LIN {X 0,Y 121.489,Z 909.455,A -85,B 0,C 180,E1 27726.454,E2 27726.454} C_VEL
LIN {X 0,Y 85.535,Z 923.158,A -85,B 0,C 180,E1 27734,E2 27734} C_VEL
LIN {X 0,Y 52.423,Z 931.161,A -85,B 0,C 180,E1 27750.283,E2 27750.283} C_VEL
LIN {X 0,Y 33.25,Z 933.945,A -85,B 0,C 180,E1 27783.011,E2 27783.011} C_VEL
LIN {X 0,Y 33.264,Z 933.922,A -85,B 0,C 180,E1 27836.977,E2 27836.977} C_VEL
LIN {X 0,Y 58.65,Z 929.923,A -85,B 0,C 180,E1 27874.226,E2 27874.226} C_VEL
LIN {X 0,Y 92.609,Z 920.78,A -85,B 0,C 180,E1 27887.866,E2 27887.866} C_VEL
LIN {X 0,Y 124.559,Z 907.865,A -85,B 0,C 180,E1 27894.091,E2 27894.091} C_VEL
LIN {X 0,Y 86.399,Z 925.528,A -85,B 0,C 180,E1 27900.019,E2 27900.019} C_VEL
LIN {X 0,Y 54.099,Z 936.193,A -85,B 0,C 180,E1 27912.507,E2 27912.507} C_VEL
LIN {X 0,Y 28.099,Z 942.904,A -85,B 0,C 180,E1 27957.519,E2 27957.519} C_VEL
LIN {X 0,Y 26.517,Z 943.563,A -85,B 0,C 180,E1 27977.697,E2 27977.697} C_VEL
LIN {X 0,Y 24.613,Z 943.517,A -85,B 0,C 180,E1 27992.94,E2 27992.94} C_VEL
LIN {X 0,Y 21.913,Z 941.506,A -85,B 0,C 180,E1 28035.111,E2 28035.111} C_VEL
LIN {X 0,Y 52.923,Z 934.846,A -85,B 0,C 180,E1 28076.336,E2 28076.336} C_VEL
LIN {X 0,Y 91.062,Z 922.515,A -85,B 0,C 180,E1 28086.143,E2 28086.143} C_VEL
LIN {X 0,Y 91.268,Z 922.217,A -85,B 0,C 180,E1 28087.247,E2 28087.247} C_VEL
LIN {X 0,Y 55.679,Z 931.309,A -85,B 0,C 180,E1 28098.458,E2 28098.458} C_VEL
LIN {X 0,Y 26.544,Z 935.256,A -85,B 0,C 180,E1 28135.356,E2 28135.356} C_VEL
LIN {X 0,Y 26.557,Z 935.233,A -85,B 0,C 180,E1 28204.625,E2 28204.625} C_VEL
LIN {X 0,Y 55.691,Z 931.242,A -85,B 0,C 180,E1 28241.506,E2 28241.506} C_VEL
LIN {X 0,Y 91.285,Z 922.099,A -85,B 0,C 180,E1 28252.673,E2 28252.673} C_VEL
LIN {X 0,Y 91.061,Z 922.421,A -85,B 0,C 180,E1 28253.867,E2 28253.867} C_VEL
LIN {X 0,Y 52.923,Z 934.79,A -85,B 0,C 180,E1 28263.671,E2 28263.671} C_VEL
LIN {X 0,Y 21.684,Z 941.535,A -85,B 0,C 180,E1 28305.9,E2 28305.9} C_VEL
LIN {X 0,Y 19.235,Z 942.611,A -85,B 0,C 180,E1 28350,E2 28350} C_VEL
LIN {X 0,Y 21.913,Z 941.506,A -85,B 0,C 180,E1 28395.111,E2 28395.111} C_VEL
LIN {X 0,Y 28.591,Z 939.62,A -85,B 0,C 180,E1 28420.824,E2 28420.824} C_VEL
LIN {X 0,Y 43.222,Z 935.698,A -85,B 0,C 180,E1 28441.962,E2 28441.962} C_VEL
LIN {X 0,Y 45.265,Z 935.239,A -85,B 0,C 180,E1 28442.871,E2 28442.871} C_VEL
LIN {X 0,Y 60.829,Z 931.445,A -85,B 0,C 180,E1 28447.124,E2 28447.124} C_VEL
LIN {X 0,Y 60.982,Z 931.252,A -85,B 0,C 180,E1 28448.195,E2 28448.195} C_VEL
LIN {X 0,Y 32.698,Z 935.56,A -85,B 0,C 180,E1 28462.632,E2 28462.632} C_VEL
LIN {X 0,Y 14.451,Z 936.94,A -85,B 0,C 180,E1 28530,E2 28530} C_VEL
LIN {X 0,Y 32.705,Z 935.522,A -85,B 0,C 180,E1 28597.338,E2 28597.338} C_VEL
LIN {X 0,Y 60.991,Z 931.186,A -85,B 0,C 180,E1 28611.75,E2 28611.75} C_VEL
LIN {X 0,Y 60.826,Z 931.393,A -85,B 0,C 180,E1 28612.9,E2 28612.9} C_VEL
LIN {X 0,Y 23.216,Z 939.266,A -85,B 0,C 180,E1 28632.841,E2 28632.841} C_VEL
LIN {X 0,Y 11.204,Z 941.259,A -85,B 0,C 180,E1 28710,E2 28710} C_VEL
LIN {X 0,Y 30.317,Z 938.164,A -85,B 0,C 180,E1 28794.537,E2 28794.537} C_VEL
LIN {X 0,Y 45.265,Z 935.239,A -85,B 0,C 180,E1 28802.871,E2 28802.871} C_VEL
LIN {X 0,Y 39.983,Z 935.649,A -85,B 0,C 180,E1 28807.386,E2 28807.386} C_VEL
LIN {X 0,Y 12.03,Z 938,A -85,B 0,C 180,E1 28832.055,E2 28832.055} C_VEL
LIN {X 0,Y 16.337,Z 937.859,A -85,B 0,C 180,E1 28957.464,E2 28957.464} C_VEL
LIN {X 0,Y 24.424,Z 937.703,A -85,B 0,C 180,E1 28971.759,E2 28971.759} C_VEL
LIN {X 0,Y 3.181,Z 939.909,A -85,B 0,C 180,E1 29069.999,E2 29069.999} C_VEL
LIN {X 0,Y 24.458,Z 937.723,A -85,B 0,C 180,E1 29168.195,E2 29168.195} C_VEL
LIN {X 0,Y 16.333,Z 937.88,A -85,B 0,C 180,E1 29182.497,E2 29182.497} C_VEL
LIN {X 0,Y 12.03,Z 938,A -85,B 0,C 180,E1 29192.055,E2 29192.055} C_VEL
LIN {X 0,Y 10.461,Z 940,A -85,B 0,C 180,E1 29197.984,E2 29197.984} C_VEL
LIN {X 0,Y 10.461,Z 1015.5,A -85,B 0,C 180,E1 29197.984,E2 29197.984} C_VEL
LIN {X 0,Y 10.461,Z 1015.5,A -85,B 0,C 180,E1 29197.984,E2 29197.984}

QRS_NEXT_CUT()
PTP {E1 29336.846,E2 29336.846}
PTP {X 0,Y 607.911,A -85,B 0,C 180,E1 29336.846,E2 29336.846,E3 0,E4 0,E5 0,E6 0}
QRS_SPEED_INIT()
LIN {X 0,Y 607.911,Z 1015.5,A -85,B 0,C 180,E1 29336.846,E2 29336.846,E3 0,E4 0,E5 0,E6 0} C_VEL
LIN {X 0,Y 607.911,Z 365.088,A -85,B 0,C 180,E1 29336.846,E2 29336.846} C_VEL
LIN {X 0,Y 607.911,Z 357.012,A -85,B 0,C 180,E1 29336.846,E2 29336.846} C_VEL
LIN {X 0,Y 607.884,Z 355.012,A -85,B 0,C 180,E1 29336.657,E2 29336.657} C_VEL
LIN {X 0,Y 607.842,Z 355.013,A -85,B 0,C 180,E1 29333.767,E2 29333.767} C_VEL
LIN {X 0,Y 607.909,Z 355.01,A -85,B 0,C 180,E1 29330.629,E2 29330.629} C_VEL
LIN {X 0,Y 607.846,Z 355.012,A -85,B 0,C 180,E1 29327.652,E2 29327.652} C_VEL
LIN {X 0,Y 607.919,Z 355.009,A -85,B 0,C 180,E1 29324.516,E2 29324.516} C_VEL
LIN {X 0,Y 607.851,Z 355.012,A -85,B 0,C 180,E1 29321.49,E2 29321.49} C_VEL
LIN {X 0,Y 607.914,Z 355.01,A -85,B 0,C 180,E1 29318.382,E2 29318.382} C_VEL
LIN {X 0,Y 607.855,Z 355.012,A -85,B 0,C 180,E1 29315.304,E2 29315.304} C_VEL
LIN {X 0,Y 607.916,Z 355.01,A -85,B 0,C 180,E1 29312.223,E2 29312.223} C_VEL
LIN {X 0,Y 607.86,Z 355.011,A -85,B 0,C 180,E1 29309.153,E2 29309.153} C_VEL
LIN {X 0,Y 607.912,Z 355.011,A -85,B 0,C 180,E1 29306.112,E2 29306.112} C_VEL
LIN {X 0,Y 607.864,Z 355.01,A -85,B 0,C 180,E1 29303.065,E2 29303.065} C_VEL
LIN {X 0,Y 607.911,Z 355.011,A -85,B 0,C 180,E1 29299.977,E2 29299.977} C_VEL
LIN {X 0,Y 607.869,Z 355.01,A -85,B 0,C 180,E1 29296.822,E2 29296.822} C_VEL
LIN {X 0,Y 607.912,Z 355.011,A -85,B 0,C 180,E1 29293.776,E2 29293.776} C_VEL
LIN {X 0,Y 607.873,Z 355.009,A -85,B 0,C 180,E1 29290.639,E2 29290.639} C_VEL
LIN {X 0,Y 607.911,Z 355.008,A -85,B 0,C 180,E1 29287.48,E2 29287.48} C_VEL
LIN {X 0,Y 607.878,Z 355.011,A -85,B 0,C 180,E1 29284.34,E2 29284.34} C_VEL
LIN {X 0,Y 607.911,Z 355.004,A -85,B 0,C 180,E1 29281.201,E2 29281.201} C_VEL
LIN {X 0,Y 607.906,Z 355.317,A -85,B 0,C 180,E1 29279.834,E2 29279.834} C_VEL
LIN {X 0,Y 607.918,Z 382.895,A -85,B 0,C 180,E1 29277.643,E2 29277.643} C_VEL
LIN {X 0,Y 607.919,Z 590.082,A -85,B 0,C 180,E1 29274.95,E2 29274.95} C_VEL
LIN {X 0,Y 607.915,Z 644.717,A -85,B 0,C 180,E1 29274.225,E2 29274.225} C_VEL
LIN {X 0,Y 607.905,Z 665.586,A -85,B 0,C 180,E1 29273.761,E2 29273.761} C_VEL
LIN {X 0,Y 607.913,Z 684.825,A -85,B 0,C 180,E1 29273.16,E2 29273.16} C_VEL
LIN {X 0,Y 607.91,Z 704.295,A -85,B 0,C 180,E1 29272.378,E2 29272.378} C_VEL
LIN {X 0,Y 607.918,Z 722.621,A -85,B 0,C 180,E1 29271.468,E2 29271.468} C_VEL
LIN {X 0,Y 607.917,Z 740.995,A -85,B 0,C 180,E1 29270.364,E2 29270.364} C_VEL
LIN {X 0,Y 607.913,Z 759.159,A -85,B 0,C 180,E1 29269.053,E2 29269.053} C_VEL
LIN {X 0,Y 607.918,Z 775.938,A -85,B 0,C 180,E1 29267.613,E2 29267.613} C_VEL
LIN {X 0,Y 607.909,Z 791.465,A -85,B 0,C 180,E1 29266.039,E2 29266.039} C_VEL
LIN {X 0,Y 607.916,Z 805.424,A -85,B 0,C 180,E1 29264.362,E2 29264.362} C_VEL
LIN {X 0,Y 607.915,Z 817.506,A -85,B 0,C 180,E1 29262.634,E2 29262.634} C_VEL
LIN {X 0,Y 607.905,Z 827.625,A -85,B 0,C 180,E1 29260.902,E2 29260.902} C_VEL
LIN {X 0,Y 607.901,Z 836.374,A -85,B 0,C 180,E1 29259.084,E2 29259.084} C_VEL
LIN {X 0,Y 607.9,Z 843.351,A -85,B 0,C 180,E1 29257.275,E2 29257.275} C_VEL
LIN {X 0,Y 607.901,Z 848.889,A -85,B 0,C 180,E1 29255.379,E2 29255.379} C_VEL
LIN {X 0,Y 607.9,Z 852.665,A -85,B 0,C 180,E1 29253.488,E2 29253.488} C_VEL
LIN {X 0,Y 607.903,Z 854.841,A -85,B 0,C 180,E1 29251.602,E2 29251.602} C_VEL
LIN {X 0,Y 607.904,Z 855.45,A -85,B 0,C 180,E1 29249.717,E2 29249.717} C_VEL
LIN {X 0,Y 607.913,Z 854.498,A -85,B 0,C 180,E1 29247.832,E2 29247.832} C_VEL
LIN {X 0,Y 607.916,Z 851.71,A -85,B 0,C 180,E1 29245.85,E2 29245.85} C_VEL
LIN {X 0,Y 607.916,Z 847.356,A -85,B 0,C 180,E1 29243.958,E2 29243.958} C_VEL
LIN {X 0,Y 607.912,Z 841.288,A -85,B 0,C 180,E1 29242.059,E2 29242.059} C_VEL
LIN {X 0,Y 607.907,Z 833.818,A -85,B 0,C 180,E1 29240.247,E2 29240.247} C_VEL
LIN {X 0,Y 607.904,Z 824.477,A -85,B 0,C 180,E1 29238.425,E2 29238.425} C_VEL
LIN {X 0,Y 607.905,Z 813.618,A -85,B 0,C 180,E1 29236.688,E2 29236.688} C_VEL
LIN {X 0,Y 607.911,Z 801.351,A -85,B 0,C 180,E1 29235.036,E2 29235.036} C_VEL
LIN {X 0,Y 607.918,Z 787.678,A -85,B 0,C 180,E1 29233.47,E2 29233.47} C_VEL
LIN {X 0,Y 607.912,Z 772.518,A -85,B 0,C 180,E1 29231.99,E2 29231.99} C_VEL
LIN {X 0,Y 607.918,Z 755.721,A -85,B 0,C 180,E1 29230.597,E2 29230.597} C_VEL
LIN {X 0,Y 607.917,Z 738.595,A -85,B 0,C 180,E1 29229.394,E2 29229.394} C_VEL
LIN {X 0,Y 607.918,Z 720.445,A -85,B 0,C 180,E1 29228.322,E2 29228.322} C_VEL
LIN {X 0,Y 607.914,Z 701.781,A -85,B 0,C 180,E1 29227.418,E2 29227.418} C_VEL
LIN {X 0,Y 607.914,Z 682.685,A -85,B 0,C 180,E1 29226.676,E2 29226.676} C_VEL
LIN {X 0,Y 607.906,Z 661.895,A -85,B 0,C 180,E1 29226.058,E2 29226.058} C_VEL
LIN {X 0,Y 607.914,Z 642.161,A -85,B 0,C 180,E1 29225.645,E2 29225.645} C_VEL
LIN {X 0,Y 607.916,Z 383.636,A -85,B 0,C 180,E1 29222.289,E2 29222.289} C_VEL
LIN {X 0,Y 607.918,Z 379.216,A -85,B 0,C 180,E1 29221.988,E2 29221.988} C_VEL
LIN {X 0,Y 607.906,Z 355.369,A -85,B 0,C 180,E1 29220.088,E2 29220.088} C_VEL
LIN {X 0,Y 607.885,Z 355.008,A -85,B 0,C 180,E1 29219.674,E2 29219.674} C_VEL
LIN {X 0,Y 607.906,Z 355.01,A -85,B 0,C 180,E1 29216.501,E2 29216.501} C_VEL
LIN {X 0,Y 607.881,Z 355.009,A -85,B 0,C 180,E1 29213.387,E2 29213.387} C_VEL
LIN {X 0,Y 607.908,Z 355.011,A -85,B 0,C 180,E1 29210.227,E2 29210.227} C_VEL
LIN {X 0,Y 607.876,Z 355.009,A -85,B 0,C 180,E1 29207.189,E2 29207.189} C_VEL
LIN {X 0,Y 607.911,Z 355.011,A -85,B 0,C 180,E1 29204.054,E2 29204.054} C_VEL
LIN {X 0,Y 607.875,Z 355.009,A -85,B 0,C 180,E1 29200.893,E2 29200.893} C_VEL
LIN {X 0,Y 607.917,Z 355.013,A -85,B 0,C 180,E1 29197.717,E2 29197.717} C_VEL
LIN {X 0,Y 607.875,Z 355.008,A -85,B 0,C 180,E1 29194.574,E2 29194.574} C_VEL
LIN {X 0,Y 607.892,Z 355.013,A -85,B 0,C 180,E1 29191.316,E2 29191.316} C_VEL
LIN {X 0,Y 607.88,Z 355.008,A -85,B 0,C 180,E1 29188.276,E2 29188.276} C_VEL
LIN {X 0,Y 607.875,Z 355.013,A -85,B 0,C 180,E1 29185.007,E2 29185.007} C_VEL
LIN {X 0,Y 607.892,Z 355.008,A -85,B 0,C 180,E1 29181.94,E2 29181.94} C_VEL
LIN {X 0,Y 607.863,Z 355.012,A -85,B 0,C 180,E1 29178.709,E2 29178.709} C_VEL
LIN {X 0,Y 607.889,Z 355.009,A -85,B 0,C 180,E1 29175.747,E2 29175.747} C_VEL
LIN {X 0,Y 607.858,Z 355.013,A -85,B 0,C 180,E1 29172.54,E2 29172.54} C_VEL
LIN {X 0,Y 607.874,Z 355.01,A -85,B 0,C 180,E1 29169.659,E2 29169.659} C_VEL
LIN {X 0,Y 607.856,Z 355.013,A -85,B 0,C 180,E1 29166.422,E2 29166.422} C_VEL
LIN {X 0,Y 607.86,Z 355.011,A -85,B 0,C 180,E1 29163.584,E2 29163.584} C_VEL
LIN {X 0,Y 607.853,Z 355.014,A -85,B 0,C 180,E1 29160.283,E2 29160.283} C_VEL
LIN {X 0,Y 607.845,Z 355.012,A -85,B 0,C 180,E1 29157.549,E2 29157.549} C_VEL
LIN {X 0,Y 607.864,Z 355.014,A -85,B 0,C 180,E1 29154.299,E2 29154.299} C_VEL
LIN {X 0,Y 607.834,Z 355.014,A -85,B 0,C 180,E1 29151.487,E2 29151.487} C_VEL
LIN {X 0,Y 607.898,Z 355.015,A -85,B 0,C 180,E1 29148.424,E2 29148.424} C_VEL
LIN {X 0,Y 607.825,Z 355.014,A -85,B 0,C 180,E1 29145.521,E2 29145.521} C_VEL
LIN {X 0,Y 607.895,Z 355.015,A -85,B 0,C 180,E1 29142.532,E2 29142.532} C_VEL
LIN {X 0,Y 607.826,Z 355.015,A -85,B 0,C 180,E1 29139.49,E2 29139.49} C_VEL
LIN {X 0,Y 607.862,Z 355.014,A -85,B 0,C 180,E1 29136.646,E2 29136.646} C_VEL
LIN {X 0,Y 607.837,Z 355.014,A -85,B 0,C 180,E1 29133.422,E2 29133.422} C_VEL
LIN {X 0,Y 607.85,Z 355.014,A -85,B 0,C 180,E1 29130.648,E2 29130.648} C_VEL
LIN {X 0,Y 607.849,Z 355.013,A -85,B 0,C 180,E1 29127.349,E2 29127.349} C_VEL
LIN {X 0,Y 607.846,Z 355.013,A -85,B 0,C 180,E1 29124.619,E2 29124.619} C_VEL
LIN {X 0,Y 607.871,Z 355.011,A -85,B 0,C 180,E1 29121.373,E2 29121.373} C_VEL
LIN {X 0,Y 607.85,Z 355.013,A -85,B 0,C 180,E1 29118.479,E2 29118.479} C_VEL
LIN {X 0,Y 607.883,Z 355.011,A -85,B 0,C 180,E1 29115.253,E2 29115.253} C_VEL
LIN {X 0,Y 607.851,Z 355.012,A -85,B 0,C 180,E1 29112.391,E2 29112.391} C_VEL
LIN {X 0,Y 607.907,Z 355.002,A -85,B 0,C 180,E1 29109.224,E2 29109.224} C_VEL
LIN {X 0,Y 607.887,Z 355.304,A -85,B 0,C 180,E1 29107.84,E2 29107.84} C_VEL
LIN {X 0,Y 607.91,Z 357.762,A -85,B 0,C 180,E1 29107.654,E2 29107.654} C_VEL
LIN {X 0,Y 607.893,Z 409.406,A -85,B 0,C 180,E1 29104.798,E2 29104.798} C_VEL
LIN {X 0,Y 607.913,Z 454.921,A -85,B 0,C 180,E1 29102.376,E2 29102.376} C_VEL
LIN {X 0,Y 607.913,Z 679.75,A -85,B 0,C 180,E1 29099.342,E2 29099.342} C_VEL
LIN {X 0,Y 607.9,Z 760.832,A -85,B 0,C 180,E1 29098.245,E2 29098.245} C_VEL
LIN {X 0,Y 607.906,Z 781.277,A -85,B 0,C 180,E1 29097.804,E2 29097.804} C_VEL
LIN {X 0,Y 607.908,Z 801.875,A -85,B 0,C 180,E1 29097.207,E2 29097.207} C_VEL
LIN {X 0,Y 607.904,Z 822.631,A -85,B 0,C 180,E1 29096.415,E2 29096.415} C_VEL
LIN {X 0,Y 607.918,Z 843.787,A -85,B 0,C 180,E1 29095.419,E2 29095.419} C_VEL
LIN {X 0,Y 607.916,Z 863.097,A -85,B 0,C 180,E1 29094.332,E2 29094.332} C_VEL
LIN {X 0,Y 607.915,Z 881.589,A -85,B 0,C 180,E1 29093.094,E2 29093.094} C_VEL
LIN {X 0,Y 607.911,Z 899.77,A -85,B 0,C 180,E1 29091.678,E2 29091.678} C_VEL
LIN {X 0,Y 607.912,Z 916.668,A -85,B 0,C 180,E1 29090.154,E2 29090.154} C_VEL
LIN {X 0,Y 607.918,Z 932.477,A -85,B 0,C 180,E1 29088.506,E2 29088.506} C_VEL
LIN {X 0,Y 607.916,Z 946.401,A -85,B 0,C 180,E1 29086.818,E2 29086.818} C_VEL
LIN {X 0,Y 607.919,Z 958.909,A -85,B 0,C 180,E1 29085.061,E2 29085.061} C_VEL
LIN {X 0,Y 607.917,Z 970.422,A -85,B 0,C 180,E1 29083.176,E2 29083.176} C_VEL
LIN {X 0,Y 607.903,Z 980.064,A -85,B 0,C 180,E1 29081.286,E2 29081.286} C_VEL
LIN {X 0,Y 607.896,Z 988.387,A -85,B 0,C 180,E1 29079.296,E2 29079.296} C_VEL
LIN {X 0,Y 607.891,Z 994.96,A -85,B 0,C 180,E1 29077.339,E2 29077.339} C_VEL
LIN {X 0,Y 607.9,Z 999.809,A -85,B 0,C 180,E1 29075.379,E2 29075.379} C_VEL
LIN {X 0,Y 607.913,Z 1003.346,A -85,B 0,C 180,E1 29073.29,E2 29073.29} C_VEL
LIN {X 0,Y 607.911,Z 1005.21,A -85,B 0,C 180,E1 29071.225,E2 29071.225} C_VEL
LIN {X 0,Y 607.895,Z 1005.329,A -85,B 0,C 180,E1 29069.246,E2 29069.246} C_VEL
LIN {X 0,Y 607.89,Z 1003.896,A -85,B 0,C 180,E1 29067.172,E2 29067.172} C_VEL
LIN {X 0,Y 607.901,Z 1001.146,A -85,B 0,C 180,E1 29065.284,E2 29065.284} C_VEL
LIN {X 0,Y 607.916,Z 996.655,A -85,B 0,C 180,E1 29063.295,E2 29063.295} C_VEL
LIN {X 0,Y 607.908,Z 990.597,A -85,B 0,C 180,E1 29061.298,E2 29061.298} C_VEL
LIN {X 0,Y 607.908,Z 983.069,A -85,B 0,C 180,E1 29059.386,E2 29059.386} C_VEL
LIN {X 0,Y 607.909,Z 973.335,A -85,B 0,C 180,E1 29057.366,E2 29057.366} C_VEL
LIN {X 0,Y 607.916,Z 962.756,A -85,B 0,C 180,E1 29055.524,E2 29055.524} C_VEL
LIN {X 0,Y 607.913,Z 950.048,A -85,B 0,C 180,E1 29053.667,E2 29053.667} C_VEL
LIN {X 0,Y 607.905,Z 935.884,A -85,B 0,C 180,E1 29051.891,E2 29051.891} C_VEL
LIN {X 0,Y 607.909,Z 920.092,A -85,B 0,C 180,E1 29050.185,E2 29050.185} C_VEL
LIN {X 0,Y 607.914,Z 903.526,A -85,B 0,C 180,E1 29048.638,E2 29048.638} C_VEL
LIN {X 0,Y 607.916,Z 885.833,A -85,B 0,C 180,E1 29047.214,E2 29047.214} C_VEL
LIN {X 0,Y 607.915,Z 867.976,A -85,B 0,C 180,E1 29045.982,E2 29045.982} C_VEL
LIN {X 0,Y 607.918,Z 848.77,A -85,B 0,C 180,E1 29044.842,E2 29044.842} C_VEL
LIN {X 0,Y 607.899,Z 829.889,A -85,B 0,C 180,E1 29043.902,E2 29043.902} C_VEL
LIN {X 0,Y 607.916,Z 809.129,A -85,B 0,C 180,E1 29043.055,E2 29043.055} C_VEL
LIN {X 0,Y 607.914,Z 789.268,A -85,B 0,C 180,E1 29042.404,E2 29042.404} C_VEL
LIN {X 0,Y 607.898,Z 769.086,A -85,B 0,C 180,E1 29041.916,E2 29041.916} C_VEL
LIN {X 0,Y 607.908,Z 747.7,A -85,B 0,C 180,E1 29041.555,E2 29041.555} C_VEL
LIN {X 0,Y 607.893,Z 527.192,A -85,B 0,C 180,E1 29038.61,E2 29038.61} C_VEL
LIN {X 0,Y 607.916,Z 454.054,A -85,B 0,C 180,E1 29037.594,E2 29037.594} C_VEL
LIN {X 0,Y 607.917,Z 396.559,A -85,B 0,C 180,E1 29034.502,E2 29034.502} C_VEL
LIN {X 0,Y 607.895,Z 355.759,A -85,B 0,C 180,E1 29032.221,E2 29032.221} C_VEL
LIN {X 0,Y 607.875,Z 355.045,A -85,B 0,C 180,E1 29032.041,E2 29032.041} C_VEL
LIN {X 0,Y 607.864,Z 355.011,A -85,B 0,C 180,E1 29029.112,E2 29029.112} C_VEL
LIN {X 0,Y 607.864,Z 355.014,A -85,B 0,C 180,E1 29025.785,E2 29025.785} C_VEL
LIN {X 0,Y 607.859,Z 355.011,A -85,B 0,C 180,E1 29022.92,E2 29022.92} C_VEL
LIN {X 0,Y 607.863,Z 355.014,A -85,B 0,C 180,E1 29019.658,E2 29019.658} C_VEL
LIN {X 0,Y 607.846,Z 355.012,A -85,B 0,C 180,E1 29016.898,E2 29016.898} C_VEL
LIN {X 0,Y 607.891,Z 355.015,A -85,B 0,C 180,E1 29013.775,E2 29013.775} C_VEL
LIN {X 0,Y 607.836,Z 355.012,A -85,B 0,C 180,E1 29010.879,E2 29010.879} C_VEL
LIN {X 0,Y 607.906,Z 355.016,A -85,B 0,C 180,E1 29007.775,E2 29007.775} C_VEL
LIN {X 0,Y 607.829,Z 355.013,A -85,B 0,C 180,E1 29004.78,E2 29004.78} C_VEL
LIN {X 0,Y 607.903,Z 355.013,A -85,B 0,C 180,E1 29001.821,E2 29001.821} C_VEL
LIN {X 0,Y 607.826,Z 355.014,A -85,B 0,C 180,E1 28998.709,E2 28998.709} C_VEL
LIN {X 0,Y 607.871,Z 355.015,A -85,B 0,C 180,E1 28995.817,E2 28995.817} C_VEL
LIN {X 0,Y 607.832,Z 355.015,A -85,B 0,C 180,E1 28992.734,E2 28992.734} C_VEL
LIN {X 0,Y 607.831,Z 355.014,A -85,B 0,C 180,E1 28990.137,E2 28990.137} C_VEL
LIN {X 0,Y 607.88,Z 355.013,A -85,B 0,C 180,E1 28986.991,E2 28986.991} C_VEL
LIN {X 0,Y 607.832,Z 355.014,A -85,B 0,C 180,E1 28984.15,E2 28984.15} C_VEL
LIN {X 0,Y 607.919,Z 355.014,A -85,B 0,C 180,E1 28981.131,E2 28981.131} C_VEL
LIN {X 0,Y 607.838,Z 355.013,A -85,B 0,C 180,E1 28978.114,E2 28978.114} C_VEL
LIN {X 0,Y 607.884,Z 355.012,A -85,B 0,C 180,E1 28976.657,E2 28976.657} C_VEL
LIN {X 0,Y 606.825,Z 355.143,A -85,B 0,C 180,E1 28975.931,E2 28975.931} C_VEL
LIN {X 0,Y 600.412,Z 355.94,A -85,B 0,C 180,E1 28973.894,E2 28973.894} C_VEL
LIN {X 0,Y 599.929,Z 356.002,A -85,B 0,C 180,E1 28973.364,E2 28973.364} C_VEL
LIN {X 0,Y 599.915,Z 356,A -85,B 0,C 180,E1 28970.115,E2 28970.115} C_VEL
LIN {X 0,Y 599.924,Z 356.003,A -85,B 0,C 180,E1 28967.291,E2 28967.291} C_VEL
LIN {X 0,Y 599.927,Z 355.999,A -85,B 0,C 180,E1 28964.038,E2 28964.038} C_VEL
LIN {X 0,Y 599.928,Z 356.002,A -85,B 0,C 180,E1 28961.136,E2 28961.136} C_VEL
LIN {X 0,Y 599.933,Z 355.998,A -85,B 0,C 180,E1 28957.873,E2 28957.873} C_VEL
LIN {X 0,Y 599.932,Z 356.002,A -85,B 0,C 180,E1 28954.955,E2 28954.955} C_VEL
LIN {X 0,Y 599.932,Z 355.998,A -85,B 0,C 180,E1 28951.628,E2 28951.628} C_VEL
LIN {X 0,Y 599.958,Z 356.002,A -85,B 0,C 180,E1 28948.558,E2 28948.558} C_VEL
LIN {X 0,Y 599.932,Z 355.998,A -85,B 0,C 180,E1 28945.367,E2 28945.367} C_VEL
LIN {X 0,Y 599.972,Z 356.003,A -85,B 0,C 180,E1 28942.294,E2 28942.294} C_VEL
LIN {X 0,Y 599.931,Z 355.998,A -85,B 0,C 180,E1 28939.081,E2 28939.081} C_VEL
LIN {X 0,Y 599.975,Z 355.999,A -85,B 0,C 180,E1 28935.905,E2 28935.905} C_VEL
LIN {X 0,Y 599.934,Z 355.999,A -85,B 0,C 180,E1 28932.835,E2 28932.835} C_VEL
LIN {X 0,Y 599.974,Z 356.002,A -85,B 0,C 180,E1 28929.782,E2 28929.782} C_VEL
LIN {X 0,Y 599.937,Z 355.997,A -85,B 0,C 180,E1 28926.625,E2 28926.625} C_VEL
LIN {X 0,Y 599.97,Z 356.001,A -85,B 0,C 180,E1 28923.474,E2 28923.474} C_VEL
LIN {X 0,Y 599.948,Z 356.054,A -85,B 0,C 180,E1 28920.312,E2 28920.312} C_VEL
LIN {X 0,Y 600.063,Z 356.688,A -85,B 0,C 180,E1 28920.141,E2 28920.141} C_VEL
LIN {X 0,Y 600.588,Z 359.133,A -85,B 0,C 180,E1 28919.904,E2 28919.904} C_VEL
LIN {X 0,Y 600.567,Z 383.206,A -85,B 0,C 180,E1 28917.998,E2 28917.998} C_VEL
LIN {X 0,Y 600.82,Z 389.233,A -85,B 0,C 180,E1 28917.897,E2 28917.897} C_VEL
LIN {X 0,Y 600.615,Z 644.031,A -85,B 0,C 180,E1 28914.551,E2 28914.551} C_VEL
LIN {X 0,Y 600.559,Z 664.328,A -85,B 0,C 180,E1 28914.102,E2 28914.102} C_VEL
LIN {X 0,Y 600.503,Z 683.819,A -85,B 0,C 180,E1 28913.499,E2 28913.499} C_VEL
LIN {X 0,Y 600.422,Z 703.775,A -85,B 0,C 180,E1 28912.697,E2 28912.697} C_VEL
LIN {X 0,Y 600.356,Z 721.813,A -85,B 0,C 180,E1 28911.799,E2 28911.799} C_VEL
LIN {X 0,Y 600.284,Z 740.392,A -85,B 0,C 180,E1 28910.675,E2 28910.675} C_VEL
LIN {X 0,Y 600.201,Z 757.787,A -85,B 0,C 180,E1 28909.414,E2 28909.414} C_VEL
LIN {X 0,Y 600.125,Z 773.738,A -85,B 0,C 180,E1 28908.05,E2 28908.05} C_VEL
LIN {X 0,Y 600.068,Z 788.696,A -85,B 0,C 180,E1 28906.552,E2 28906.552} C_VEL
LIN {X 0,Y 600.014,Z 802.199,A -85,B 0,C 180,E1 28904.967,E2 28904.967} C_VEL
LIN {X 0,Y 599.967,Z 814.393,A -85,B 0,C 180,E1 28903.282,E2 28903.282} C_VEL
LIN {X 0,Y 599.939,Z 825.039,A -85,B 0,C 180,E1 28901.535,E2 28901.535} C_VEL
LIN {X 0,Y 599.925,Z 834.312,A -85,B 0,C 180,E1 28899.689,E2 28899.689} C_VEL
LIN {X 0,Y 599.919,Z 841.666,A -85,B 0,C 180,E1 28897.854,E2 28897.854} C_VEL
LIN {X 0,Y 599.917,Z 847.625,A -85,B 0,C 180,E1 28895.93,E2 28895.93} C_VEL
LIN {X 0,Y 599.917,Z 851.877,A -85,B 0,C 180,E1 28894.013,E2 28894.013} C_VEL
LIN {X 0,Y 599.915,Z 854.503,A -85,B 0,C 180,E1 28892.101,E2 28892.101} C_VEL
LIN {X 0,Y 599.912,Z 855.474,A -85,B 0,C 180,E1 28890.095,E2 28890.095} C_VEL
LIN {X 0,Y 599.909,Z 854.771,A -85,B 0,C 180,E1 28888.185,E2 28888.185} C_VEL
LIN {X 0,Y 599.913,Z 852.341,A -85,B 0,C 180,E1 28886.177,E2 28886.177} C_VEL
LIN {X 0,Y 599.918,Z 848.115,A -85,B 0,C 180,E1 28884.165,E2 28884.165} C_VEL
LIN {X 0,Y 599.925,Z 842.347,A -85,B 0,C 180,E1 28882.242,E2 28882.242} C_VEL
LIN {X 0,Y 599.928,Z 834.718,A -85,B 0,C 180,E1 28880.31,E2 28880.31} C_VEL
LIN {X 0,Y 599.939,Z 825.513,A -85,B 0,C 180,E1 28878.464,E2 28878.464} C_VEL
LIN {X 0,Y 599.968,Z 814.895,A -85,B 0,C 180,E1 28876.705,E2 28876.705} C_VEL
LIN {X 0,Y 600.01,Z 802.899,A -85,B 0,C 180,E1 28875.032,E2 28875.032} C_VEL
LIN {X 0,Y 600.065,Z 789.526,A -85,B 0,C 180,E1 28873.447,E2 28873.447} C_VEL
LIN {X 0,Y 600.124,Z 774.721,A -85,B 0,C 180,E1 28871.949,E2 28871.949} C_VEL
LIN {X 0,Y 600.202,Z 758.36,A -85,B 0,C 180,E1 28870.54,E2 28870.54} C_VEL
LIN {X 0,Y 600.277,Z 740.968,A -85,B 0,C 180,E1 28869.273,E2 28869.273} C_VEL
LIN {X 0,Y 600.35,Z 722.477,A -85,B 0,C 180,E1 28868.149,E2 28868.149} C_VEL
LIN {X 0,Y 600.422,Z 704.009,A -85,B 0,C 180,E1 28867.223,E2 28867.223} C_VEL
LIN {X 0,Y 600.501,Z 684.14,A -85,B 0,C 180,E1 28866.422,E2 28866.422} C_VEL
LIN {X 0,Y 600.558,Z 664.231,A -85,B 0,C 180,E1 28865.805,E2 28865.805} C_VEL
LIN {X 0,Y 600.616,Z 644.079,A -85,B 0,C 180,E1 28865.359,E2 28865.359} C_VEL
LIN {X 0,Y 600.825,Z 387.532,A -85,B 0,C 180,E1 28861.991,E2 28861.991} C_VEL
LIN {X 0,Y 600.547,Z 383.03,A -85,B 0,C 180,E1 28861.905,E2 28861.905} C_VEL
LIN {X 0,Y 600.55,Z 358.194,A -85,B 0,C 180,E1 28859.928,E2 28859.928} C_VEL
LIN {X 0,Y 599.96,Z 356.103,A -85,B 0,C 180,E1 28859.674,E2 28859.674} C_VEL
LIN {X 0,Y 599.968,Z 356,A -85,B 0,C 180,E1 28856.525,E2 28856.525} C_VEL
LIN {X 0,Y 599.942,Z 355.997,A -85,B 0,C 180,E1 28853.374,E2 28853.374} C_VEL
LIN {X 0,Y 599.97,Z 356.001,A -85,B 0,C 180,E1 28850.198,E2 28850.198} C_VEL
LIN {X 0,Y 599.938,Z 355.998,A -85,B 0,C 180,E1 28847.163,E2 28847.163} C_VEL
LIN {X 0,Y 599.975,Z 356,A -85,B 0,C 180,E1 28843.957,E2 28843.957} C_VEL
LIN {X 0,Y 599.94,Z 355.997,A -85,B 0,C 180,E1 28840.792,E2 28840.792} C_VEL
LIN {X 0,Y 599.96,Z 356.003,A -85,B 0,C 180,E1 28837.515,E2 28837.515} C_VEL
LIN {X 0,Y 599.949,Z 355.996,A -85,B 0,C 180,E1 28834.4,E2 28834.4} C_VEL
LIN {X 0,Y 599.936,Z 356.001,A -85,B 0,C 180,E1 28831.108,E2 28831.108} C_VEL
LIN {X 0,Y 599.974,Z 355.996,A -85,B 0,C 180,E1 28827.974,E2 28827.974} C_VEL
LIN {X 0,Y 599.926,Z 356.001,A -85,B 0,C 180,E1 28824.834,E2 28824.834} C_VEL
LIN {X 0,Y 599.968,Z 355.996,A -85,B 0,C 180,E1 28821.817,E2 28821.817} C_VEL
LIN {X 0,Y 599.922,Z 356.001,A -85,B 0,C 180,E1 28818.663,E2 28818.663} C_VEL
LIN {X 0,Y 599.959,Z 355.998,A -85,B 0,C 180,E1 28815.663,E2 28815.663} C_VEL
LIN {X 0,Y 599.918,Z 356.002,A -85,B 0,C 180,E1 28812.513,E2 28812.513} C_VEL
LIN {X 0,Y 599.942,Z 355.998,A -85,B 0,C 180,E1 28809.594,E2 28809.594} C_VEL
LIN {X 0,Y 599.917,Z 356.001,A -85,B 0,C 180,E1 28806.412,E2 28806.412} C_VEL
LIN {X 0,Y 599.925,Z 356,A -85,B 0,C 180,E1 28803.536,E2 28803.536} C_VEL
LIN {X 0,Y 599.914,Z 356.003,A -85,B 0,C 180,E1 28800.287,E2 28800.287} C_VEL
LIN {X 0,Y 599.908,Z 356.001,A -85,B 0,C 180,E1 28797.517,E2 28797.517} C_VEL
LIN {X 0,Y 599.916,Z 356.003,A -85,B 0,C 180,E1 28794.213,E2 28794.213} C_VEL
LIN {X 0,Y 599.896,Z 356.003,A -85,B 0,C 180,E1 28791.47,E2 28791.47} C_VEL
LIN {X 0,Y 599.95,Z 356.004,A -85,B 0,C 180,E1 28788.366,E2 28788.366} C_VEL
LIN {X 0,Y 599.887,Z 356.003,A -85,B 0,C 180,E1 28785.423,E2 28785.423} C_VEL
LIN {X 0,Y 599.966,Z 356.004,A -85,B 0,C 180,E1 28782.344,E2 28782.344} C_VEL
LIN {X 0,Y 599.885,Z 356.004,A -85,B 0,C 180,E1 28779.308,E2 28779.308} C_VEL
LIN {X 0,Y 599.975,Z 356,A -85,B 0,C 180,E1 28776.216,E2 28776.216} C_VEL
LIN {X 0,Y 599.891,Z 356.003,A -85,B 0,C 180,E1 28773.148,E2 28773.148} C_VEL
LIN {X 0,Y 599.971,Z 356.001,A -85,B 0,C 180,E1 28770.114,E2 28770.114} C_VEL
LIN {X 0,Y 599.899,Z 356.003,A -85,B 0,C 180,E1 28767.088,E2 28767.088} C_VEL
LIN {X 0,Y 599.947,Z 356.002,A -85,B 0,C 180,E1 28764.2,E2 28764.2} C_VEL
LIN {X 0,Y 599.909,Z 356.001,A -85,B 0,C 180,E1 28761.073,E2 28761.073} C_VEL
LIN {X 0,Y 599.938,Z 356.003,A -85,B 0,C 180,E1 28758.151,E2 28758.151} C_VEL
LIN {X 0,Y 599.916,Z 356.001,A -85,B 0,C 180,E1 28754.901,E2 28754.901} C_VEL
LIN {X 0,Y 599.947,Z 356.001,A -85,B 0,C 180,E1 28751.931,E2 28751.931} C_VEL
LIN {X 0,Y 599.918,Z 355.984,A -85,B 0,C 180,E1 28748.678,E2 28748.678} C_VEL
LIN {X 0,Y 599.959,Z 356.307,A -85,B 0,C 180,E1 28748.369,E2 28748.369} C_VEL
LIN {X 0,Y 601.251,Z 359.782,A -85,B 0,C 180,E1 28748.03,E2 28748.03} C_VEL
LIN {X 0,Y 601.05,Z 411.517,A -85,B 0,C 180,E1 28745.136,E2 28745.136} C_VEL
LIN {X 0,Y 601.04,Z 455.306,A -85,B 0,C 180,E1 28742.785,E2 28742.785} C_VEL
LIN {X 0,Y 600.971,Z 648.635,A -85,B 0,C 180,E1 28740.135,E2 28740.135} C_VEL
LIN {X 0,Y 600.843,Z 761.046,A -85,B 0,C 180,E1 28738.604,E2 28738.604} C_VEL
LIN {X 0,Y 600.786,Z 782.005,A -85,B 0,C 180,E1 28738.144,E2 28738.144} C_VEL
LIN {X 0,Y 600.712,Z 802.614,A -85,B 0,C 180,E1 28737.533,E2 28737.533} C_VEL
LIN {X 0,Y 600.636,Z 822.634,A -85,B 0,C 180,E1 28736.76,E2 28736.76} C_VEL
LIN {X 0,Y 600.539,Z 843.935,A -85,B 0,C 180,E1 28735.746,E2 28735.746} C_VEL
LIN {X 0,Y 600.444,Z 863.142,A -85,B 0,C 180,E1 28734.651,E2 28734.651} C_VEL
LIN {X 0,Y 600.354,Z 881.419,A -85,B 0,C 180,E1 28733.414,E2 28733.414} C_VEL
LIN {X 0,Y 600.249,Z 899.294,A -85,B 0,C 180,E1 28732.009,E2 28732.009} C_VEL
LIN {X 0,Y 600.159,Z 916.161,A -85,B 0,C 180,E1 28730.477,E2 28730.477} C_VEL
LIN {X 0,Y 600.108,Z 931.646,A -85,B 0,C 180,E1 28728.852,E2 28728.852} C_VEL
LIN {X 0,Y 600.04,Z 945.57,A -85,B 0,C 180,E1 28727.152,E2 28727.152} C_VEL
LIN {X 0,Y 599.989,Z 958.91,A -85,B 0,C 180,E1 28725.265,E2 28725.265} C_VEL
LIN {X 0,Y 599.952,Z 970.216,A -85,B 0,C 180,E1 28723.393,E2 28723.393} C_VEL
LIN {X 0,Y 599.925,Z 979.847,A -85,B 0,C 180,E1 28721.484,E2 28721.484} C_VEL
LIN {X 0,Y 599.905,Z 988.111,A -85,B 0,C 180,E1 28719.497,E2 28719.497} C_VEL
LIN {X 0,Y 599.903,Z 994.585,A -85,B 0,C 180,E1 28717.566,E2 28717.566} C_VEL
LIN {X 0,Y 599.911,Z 999.604,A -85,B 0,C 180,E1 28715.547,E2 28715.547} C_VEL
LIN {X 0,Y 599.915,Z 1003.222,A -85,B 0,C 180,E1 28713.44,E2 28713.44} C_VEL
LIN {X 0,Y 599.901,Z 1005.081,A -85,B 0,C 180,E1 28711.433,E2 28711.433} C_VEL
LIN {X 0,Y 599.891,Z 1005.373,A -85,B 0,C 180,E1 28709.427,E2 28709.427} C_VEL
LIN {X 0,Y 599.896,Z 1004.233,A -85,B 0,C 180,E1 28707.421,E2 28707.421} C_VEL
LIN {X 0,Y 599.909,Z 1001.463,A -85,B 0,C 180,E1 28705.412,E2 28705.412} C_VEL
LIN {X 0,Y 599.92,Z 996.909,A -85,B 0,C 180,E1 28703.301,E2 28703.301} C_VEL
LIN {X 0,Y 599.919,Z 990.792,A -85,B 0,C 180,E1 28701.235,E2 28701.235} C_VEL
LIN {X 0,Y 599.927,Z 983.07,A -85,B 0,C 180,E1 28699.243,E2 28699.243} C_VEL
LIN {X 0,Y 599.949,Z 973.336,A -85,B 0,C 180,E1 28697.195,E2 28697.195} C_VEL
LIN {X 0,Y 599.988,Z 962.755,A -85,B 0,C 180,E1 28695.329,E2 28695.329} C_VEL
LIN {X 0,Y 600.025,Z 950.049,A -85,B 0,C 180,E1 28693.446,E2 28693.446} C_VEL
LIN {X 0,Y 600.075,Z 935.885,A -85,B 0,C 180,E1 28691.647,E2 28691.647} C_VEL
LIN {X 0,Y 600.156,Z 920.218,A -85,B 0,C 180,E1 28689.931,E2 28689.931} C_VEL
LIN {X 0,Y 600.241,Z 904.131,A -85,B 0,C 180,E1 28688.402,E2 28688.402} C_VEL
LIN {X 0,Y 600.32,Z 885.833,A -85,B 0,C 180,E1 28686.909,E2 28686.909} C_VEL
LIN {X 0,Y 600.421,Z 867.176,A -85,B 0,C 180,E1 28685.61,E2 28685.61} C_VEL
LIN {X 0,Y 600.533,Z 846.786,A -85,B 0,C 180,E1 28684.405,E2 28684.405} C_VEL
LIN {X 0,Y 600.599,Z 827.615,A -85,B 0,C 180,E1 28683.452,E2 28683.452} C_VEL
LIN {X 0,Y 600.701,Z 807.05,A -85,B 0,C 180,E1 28682.628,E2 28682.628} C_VEL
LIN {X 0,Y 600.787,Z 785.722,A -85,B 0,C 180,E1 28681.953,E2 28681.953} C_VEL
LIN {X 0,Y 600.821,Z 765.977,A -85,B 0,C 180,E1 28681.49,E2 28681.49} C_VEL
LIN {X 0,Y 600.89,Z 737.832,A -85,B 0,C 180,E1 28681.06,E2 28681.06} C_VEL
LIN {X 0,Y 601.063,Z 512.335,A -85,B 0,C 180,E1 28678.007,E2 28678.007} C_VEL
LIN {X 0,Y 600.998,Z 454.722,A -85,B 0,C 180,E1 28677.194,E2 28677.194} C_VEL
LIN {X 0,Y 601.118,Z 398.862,A -85,B 0,C 180,E1 28674.167,E2 28674.167} C_VEL
LIN {X 0,Y 601.214,Z 359.452,A -85,B 0,C 180,E1 28671.949,E2 28671.949} C_VEL
LIN {X 0,Y 599.958,Z 356.295,A -85,B 0,C 180,E1 28671.631,E2 28671.631} C_VEL
LIN {X 0,Y 599.977,Z 355.984,A -85,B 0,C 180,E1 28670.59,E2 28670.59} C_VEL
LIN {X 0,Y 599.911,Z 355.998,A -85,B 0,C 180,E1 28667.551,E2 28667.551} C_VEL
LIN {X 0,Y 599.976,Z 356,A -85,B 0,C 180,E1 28664.505,E2 28664.505} C_VEL
LIN {X 0,Y 599.909,Z 356.002,A -85,B 0,C 180,E1 28661.416,E2 28661.416} C_VEL
LIN {X 0,Y 599.955,Z 356,A -85,B 0,C 180,E1 28658.435,E2 28658.435} C_VEL
LIN {X 0,Y 599.904,Z 356.001,A -85,B 0,C 180,E1 28655.255,E2 28655.255} C_VEL
LIN {X 0,Y 599.941,Z 356.001,A -85,B 0,C 180,E1 28652.342,E2 28652.342} C_VEL
LIN {X 0,Y 599.901,Z 356.002,A -85,B 0,C 180,E1 28649.16,E2 28649.16} C_VEL
LIN {X 0,Y 599.918,Z 356.002,A -85,B 0,C 180,E1 28646.316,E2 28646.316} C_VEL
LIN {X 0,Y 599.901,Z 356.002,A -85,B 0,C 180,E1 28643.059,E2 28643.059} C_VEL
LIN {X 0,Y 599.904,Z 356.003,A -85,B 0,C 180,E1 28640.24,E2 28640.24} C_VEL
LIN {X 0,Y 599.9,Z 356.004,A -85,B 0,C 180,E1 28636.944,E2 28636.944} C_VEL
LIN {X 0,Y 599.893,Z 356.004,A -85,B 0,C 180,E1 28634.182,E2 28634.182} C_VEL
LIN {X 0,Y 599.919,Z 356.003,A -85,B 0,C 180,E1 28630.952,E2 28630.952} C_VEL
LIN {X 0,Y 599.891,Z 356.003,A -85,B 0,C 180,E1 28628.137,E2 28628.137} C_VEL
LIN {X 0,Y 599.96,Z 356.002,A -85,B 0,C 180,E1 28625.067,E2 28625.067} C_VEL
LIN {X 0,Y 599.895,Z 356.002,A -85,B 0,C 180,E1 28622.101,E2 28622.101} C_VEL
LIN {X 0,Y 599.978,Z 356.001,A -85,B 0,C 180,E1 28619.045,E2 28619.045} C_VEL
LIN {X 0,Y 599.9,Z 356.002,A -85,B 0,C 180,E1 28615.986,E2 28615.986} C_VEL
LIN {X 0,Y 599.929,Z 356.002,A -85,B 0,C 180,E1 28613.364,E2 28613.364} C_VEL
LIN {X 0,Y 598.992,Z 356.126,A -85,B 0,C 180,E1 28612.629,E2 28612.629} C_VEL
LIN {X 0,Y 592.432,Z 356.937,A -85,B 0,C 180,E1 28610.512,E2 28610.512} C_VEL
LIN {X 0,Y 591.972,Z 356.988,A -85,B 0,C 180,E1 28610.027,E2 28610.027} C_VEL
LIN {X 0,Y 592.003,Z 356.992,A -85,B 0,C 180,E1 28607.118,E2 28607.118} C_VEL
LIN {X 0,Y 591.98,Z 356.989,A -85,B 0,C 180,E1 28603.919,E2 28603.919} C_VEL
LIN {X 0,Y 592.014,Z 356.992,A -85,B 0,C 180,E1 28600.874,E2 28600.874} C_VEL
LIN {X 0,Y 591.981,Z 356.988,A -85,B 0,C 180,E1 28597.664,E2 28597.664} C_VEL
LIN {X 0,Y 592.028,Z 356.993,A -85,B 0,C 180,E1 28594.597,E2 28594.597} C_VEL
LIN {X 0,Y 591.983,Z 356.989,A -85,B 0,C 180,E1 28591.424,E2 28591.424} C_VEL
LIN {X 0,Y 592.039,Z 356.992,A -85,B 0,C 180,E1 28588.316,E2 28588.316} C_VEL
LIN {X 0,Y 591.987,Z 356.988,A -85,B 0,C 180,E1 28585.161,E2 28585.161} C_VEL
LIN {X 0,Y 592.037,Z 356.984,A -85,B 0,C 180,E1 28582.055,E2 28582.055} C_VEL
LIN {X 0,Y 591.99,Z 356.988,A -85,B 0,C 180,E1 28578.927,E2 28578.927} C_VEL
LIN {X 0,Y 592.035,Z 356.985,A -85,B 0,C 180,E1 28575.725,E2 28575.725} C_VEL
LIN {X 0,Y 591.996,Z 356.99,A -85,B 0,C 180,E1 28572.575,E2 28572.575} C_VEL
LIN {X 0,Y 592.036,Z 356.985,A -85,B 0,C 180,E1 28569.331,E2 28569.331} C_VEL
LIN {X 0,Y 592.015,Z 356.989,A -85,B 0,C 180,E1 28566.112,E2 28566.112} C_VEL
LIN {X 0,Y 592.011,Z 356.988,A -85,B 0,C 180,E1 28562.745,E2 28562.745} C_VEL
LIN {X 0,Y 592.033,Z 357.184,A -85,B 0,C 180,E1 28560.578,E2 28560.578} C_VEL
LIN {X 0,Y 593.266,Z 361.864,A -85,B 0,C 180,E1 28560.088,E2 28560.088} C_VEL
LIN {X 0,Y 593.217,Z 383.41,A -85,B 0,C 180,E1 28558.372,E2 28558.372} C_VEL
LIN {X 0,Y 593.754,Z 387.573,A -85,B 0,C 180,E1 28558.281,E2 28558.281} C_VEL
LIN {X 0,Y 593.334,Z 643.972,A -85,B 0,C 180,E1 28554.875,E2 28554.875} C_VEL
LIN {X 0,Y 593.229,Z 664.355,A -85,B 0,C 180,E1 28554.419,E2 28554.419} C_VEL
LIN {X 0,Y 593.109,Z 683.84,A -85,B 0,C 180,E1 28553.81,E2 28553.81} C_VEL
LIN {X 0,Y 592.953,Z 703.211,A -85,B 0,C 180,E1 28553.027,E2 28553.027} C_VEL
LIN {X 0,Y 592.819,Z 721.822,A -85,B 0,C 180,E1 28552.091,E2 28552.091} C_VEL
LIN {X 0,Y 592.663,Z 740.404,A -85,B 0,C 180,E1 28550.954,E2 28550.954} C_VEL
LIN {X 0,Y 592.498,Z 757.875,A -85,B 0,C 180,E1 28549.67,E2 28549.67} C_VEL
LIN {X 0,Y 592.349,Z 773.745,A -85,B 0,C 180,E1 28548.296,E2 28548.296} C_VEL
LIN {X 0,Y 592.228,Z 788.703,A -85,B 0,C 180,E1 28546.778,E2 28546.778} C_VEL
LIN {X 0,Y 592.124,Z 802.206,A -85,B 0,C 180,E1 28545.171,E2 28545.171} C_VEL
LIN {X 0,Y 592.032,Z 814.959,A -85,B 0,C 180,E1 28543.376,E2 28543.376} C_VEL
LIN {X 0,Y 591.974,Z 825.62,A -85,B 0,C 180,E1 28541.582,E2 28541.582} C_VEL
LIN {X 0,Y 591.943,Z 834.754,A -85,B 0,C 180,E1 28539.723,E2 28539.723} C_VEL
LIN {X 0,Y 591.929,Z 842.376,A -85,B 0,C 180,E1 28537.765,E2 28537.765} C_VEL
LIN {X 0,Y 591.919,Z 847.88,A -85,B 0,C 180,E1 28535.913,E2 28535.913} C_VEL
LIN {X 0,Y 591.918,Z 852.195,A -85,B 0,C 180,E1 28533.874,E2 28533.874} C_VEL
LIN {X 0,Y 591.916,Z 854.643,A -85,B 0,C 180,E1 28531.936,E2 28531.936} C_VEL
LIN {X 0,Y 591.915,Z 855.494,A -85,B 0,C 180,E1 28529.903,E2 28529.903} C_VEL
LIN {X 0,Y 591.914,Z 854.57,A -85,B 0,C 180,E1 28527.87,E2 28527.87} C_VEL
LIN {X 0,Y 591.917,Z 852.025,A -85,B 0,C 180,E1 28525.932,E2 28525.932} C_VEL
LIN {X 0,Y 591.921,Z 847.86,A -85,B 0,C 180,E1 28523.989,E2 28523.989} C_VEL
LIN {X 0,Y 591.931,Z 842.345,A -85,B 0,C 180,E1 28522.137,E2 28522.137} C_VEL
LIN {X 0,Y 591.945,Z 834.716,A -85,B 0,C 180,E1 28520.178,E2 28520.178} C_VEL
LIN {X 0,Y 591.974,Z 825.511,A -85,B 0,C 180,E1 28518.307,E2 28518.307} C_VEL
LIN {X 0,Y 592.031,Z 814.891,A -85,B 0,C 180,E1 28516.524,E2 28516.524} C_VEL
LIN {X 0,Y 592.117,Z 802.895,A -85,B 0,C 180,E1 28514.828,E2 28514.828} C_VEL
LIN {X 0,Y 592.223,Z 789.248,A -85,B 0,C 180,E1 28513.192,E2 28513.192} C_VEL
LIN {X 0,Y 592.344,Z 774.716,A -85,B 0,C 180,E1 28511.703,E2 28511.703} C_VEL
LIN {X 0,Y 592.498,Z 758.354,A -85,B 0,C 180,E1 28510.277,E2 28510.277} C_VEL
LIN {X 0,Y 592.655,Z 740.955,A -85,B 0,C 180,E1 28508.993,E2 28508.993} C_VEL
LIN {X 0,Y 592.806,Z 722.461,A -85,B 0,C 180,E1 28507.856,E2 28507.856} C_VEL
LIN {X 0,Y 592.952,Z 703.999,A -85,B 0,C 180,E1 28506.92,E2 28506.92} C_VEL
LIN {X 0,Y 593.106,Z 684.125,A -85,B 0,C 180,E1 28506.11,E2 28506.11} C_VEL
LIN {X 0,Y 593.229,Z 664.206,A -85,B 0,C 180,E1 28505.487,E2 28505.487} C_VEL
LIN {X 0,Y 593.335,Z 644.039,A -85,B 0,C 180,E1 28505.037,E2 28505.037} C_VEL
LIN {X 0,Y 593.752,Z 389.39,A -85,B 0,C 180,E1 28501.653,E2 28501.653} C_VEL
LIN {X 0,Y 593.447,Z 384.6,A -85,B 0,C 180,E1 28501.573,E2 28501.573} C_VEL
LIN {X 0,Y 593.151,Z 382.815,A -85,B 0,C 180,E1 28501.51,E2 28501.51} C_VEL
LIN {X 0,Y 593.165,Z 360.909,A -85,B 0,C 180,E1 28499.738,E2 28499.738} C_VEL
LIN {X 0,Y 592.043,Z 357.203,A -85,B 0,C 180,E1 28499.338,E2 28499.338} C_VEL
LIN {X 0,Y 592.037,Z 356.987,A -85,B 0,C 180,E1 28496.133,E2 28496.133} C_VEL
LIN {X 0,Y 592.031,Z 356.981,A -85,B 0,C 180,E1 28492.803,E2 28492.803} C_VEL
LIN {X 0,Y 592.007,Z 356.986,A -85,B 0,C 180,E1 28489.572,E2 28489.572} C_VEL
LIN {X 0,Y 592.037,Z 356.985,A -85,B 0,C 180,E1 28486.429,E2 28486.429} C_VEL
LIN {X 0,Y 591.999,Z 356.988,A -85,B 0,C 180,E1 28483.292,E2 28483.292} C_VEL
LIN {X 0,Y 592.035,Z 356.987,A -85,B 0,C 180,E1 28480.095,E2 28480.095} C_VEL
LIN {X 0,Y 591.993,Z 356.988,A -85,B 0,C 180,E1 28476.961,E2 28476.961} C_VEL
LIN {X 0,Y 592.036,Z 356.989,A -85,B 0,C 180,E1 28473.815,E2 28473.815} C_VEL
LIN {X 0,Y 591.988,Z 356.987,A -85,B 0,C 180,E1 28470.669,E2 28470.669} C_VEL
LIN {X 0,Y 592.037,Z 356.991,A -85,B 0,C 180,E1 28467.455,E2 28467.455} C_VEL
LIN {X 0,Y 591.988,Z 356.988,A -85,B 0,C 180,E1 28464.338,E2 28464.338} C_VEL
LIN {X 0,Y 592.013,Z 356.992,A -85,B 0,C 180,E1 28461.084,E2 28461.084} C_VEL
LIN {X 0,Y 591.994,Z 356.987,A -85,B 0,C 180,E1 28458.004,E2 28458.004} C_VEL
LIN {X 0,Y 591.987,Z 356.99,A -85,B 0,C 180,E1 28454.676,E2 28454.676} C_VEL
LIN {X 0,Y 592.001,Z 356.988,A -85,B 0,C 180,E1 28451.694,E2 28451.694} C_VEL
LIN {X 0,Y 591.979,Z 356.991,A -85,B 0,C 180,E1 28448.45,E2 28448.45} C_VEL
LIN {X 0,Y 591.994,Z 356.987,A -85,B 0,C 180,E1 28445.525,E2 28445.525} C_VEL
LIN {X 0,Y 591.976,Z 356.99,A -85,B 0,C 180,E1 28442.323,E2 28442.323} C_VEL
LIN {X 0,Y 591.983,Z 356.99,A -85,B 0,C 180,E1 28439.42,E2 28439.42} C_VEL
LIN {X 0,Y 591.969,Z 356.992,A -85,B 0,C 180,E1 28436.126,E2 28436.126} C_VEL
LIN {X 0,Y 591.978,Z 356.99,A -85,B 0,C 180,E1 28433.238,E2 28433.238} C_VEL
LIN {X 0,Y 591.962,Z 356.992,A -85,B 0,C 180,E1 28429.941,E2 28429.941} C_VEL
LIN {X 0,Y 591.961,Z 356.992,A -85,B 0,C 180,E1 28427.217,E2 28427.217} C_VEL
LIN {X 0,Y 591.968,Z 356.993,A -85,B 0,C 180,E1 28423.919,E2 28423.919} C_VEL
LIN {X 0,Y 591.949,Z 356.992,A -85,B 0,C 180,E1 28421.179,E2 28421.179} C_VEL
LIN {X 0,Y 591.994,Z 356.991,A -85,B 0,C 180,E1 28417.979,E2 28417.979} C_VEL
LIN {X 0,Y 591.951,Z 356.989,A -85,B 0,C 180,E1 28415.088,E2 28415.088} C_VEL
LIN {X 0,Y 592.027,Z 356.99,A -85,B 0,C 180,E1 28411.998,E2 28411.998} C_VEL
LIN {X 0,Y 591.957,Z 356.988,A -85,B 0,C 180,E1 28408.992,E2 28408.992} C_VEL
LIN {X 0,Y 592.039,Z 356.988,A -85,B 0,C 180,E1 28405.896,E2 28405.896} C_VEL
LIN {X 0,Y 591.963,Z 356.991,A -85,B 0,C 180,E1 28402.794,E2 28402.794} C_VEL
LIN {X 0,Y 592.038,Z 356.988,A -85,B 0,C 180,E1 28399.698,E2 28399.698} C_VEL
LIN {X 0,Y 591.969,Z 356.99,A -85,B 0,C 180,E1 28396.57,E2 28396.57} C_VEL
LIN {X 0,Y 592.033,Z 356.984,A -85,B 0,C 180,E1 28393.417,E2 28393.417} C_VEL
LIN {X 0,Y 591.975,Z 356.993,A -85,B 0,C 180,E1 28390.382,E2 28390.382} C_VEL
LIN {X 0,Y 592.023,Z 357.165,A -85,B 0,C 180,E1 28388.949,E2 28388.949} C_VEL
LIN {X 0,Y 592.637,Z 359.298,A -85,B 0,C 180,E1 28388.712,E2 28388.712} C_VEL
LIN {X 0,Y 594.611,Z 363.476,A -85,B 0,C 180,E1 28388.317,E2 28388.317} C_VEL
LIN {X 0,Y 594.218,Z 414.579,A -85,B 0,C 180,E1 28385.43,E2 28385.43} C_VEL
LIN {X 0,Y 594.099,Z 455.361,A -85,B 0,C 180,E1 28383.216,E2 28383.216} C_VEL
LIN {X 0,Y 594.402,Z 461.097,A -85,B 0,C 180,E1 28383.116,E2 28383.116} C_VEL
LIN {X 0,Y 593.971,Z 687.339,A -85,B 0,C 180,E1 28379.997,E2 28379.997} C_VEL
LIN {X 0,Y 593.809,Z 761.902,A -85,B 0,C 180,E1 28378.961,E2 28378.961} C_VEL
LIN {X 0,Y 593.689,Z 782.798,A -85,B 0,C 180,E1 28378.49,E2 28378.49} C_VEL
LIN {X 0,Y 593.534,Z 803.499,A -85,B 0,C 180,E1 28377.862,E2 28377.862} C_VEL
LIN {X 0,Y 593.381,Z 823.91,A -85,B 0,C 180,E1 28377.059,E2 28377.059} C_VEL
LIN {X 0,Y 593.182,Z 843.793,A -85,B 0,C 180,E1 28376.097,E2 28376.097} C_VEL
LIN {X 0,Y 593.004,Z 863.138,A -85,B 0,C 180,E1 28374.982,E2 28374.982} C_VEL
LIN {X 0,Y 592.807,Z 881.666,A -85,B 0,C 180,E1 28373.712,E2 28373.712} C_VEL
LIN {X 0,Y 592.604,Z 899.296,A -85,B 0,C 180,E1 28372.309,E2 28372.309} C_VEL
LIN {X 0,Y 592.436,Z 916.161,A -85,B 0,C 180,E1 28370.756,E2 28370.756} C_VEL
LIN {X 0,Y 592.308,Z 931.601,A -85,B 0,C 180,E1 28369.115,E2 28369.115} C_VEL
LIN {X 0,Y 592.174,Z 945.571,A -85,B 0,C 180,E1 28367.387,E2 28367.387} C_VEL
LIN {X 0,Y 592.068,Z 958.911,A -85,B 0,C 180,E1 28365.474,E2 28365.474} C_VEL
LIN {X 0,Y 592.002,Z 970.217,A -85,B 0,C 180,E1 28363.577,E2 28363.577} C_VEL
LIN {X 0,Y 591.953,Z 979.603,A -85,B 0,C 180,E1 28361.693,E2 28361.693} C_VEL
LIN {X 0,Y 591.919,Z 988.112,A -85,B 0,C 180,E1 28359.626,E2 28359.626} C_VEL
LIN {X 0,Y 591.915,Z 994.585,A -85,B 0,C 180,E1 28357.668,E2 28357.668} C_VEL
LIN {X 0,Y 591.917,Z 999.604,A -85,B 0,C 180,E1 28355.622,E2 28355.622} C_VEL
LIN {X 0,Y 591.913,Z 1003.222,A -85,B 0,C 180,E1 28353.486,E2 28353.486} C_VEL
LIN {X 0,Y 591.9,Z 1005.081,A -85,B 0,C 180,E1 28351.452,E2 28351.452} C_VEL
LIN {X 0,Y 591.891,Z 1005.373,A -85,B 0,C 180,E1 28349.42,E2 28349.42} C_VEL
LIN {X 0,Y 591.894,Z 1004.233,A -85,B 0,C 180,E1 28347.386,E2 28347.386} C_VEL
LIN {X 0,Y 591.907,Z 1001.463,A -85,B 0,C 180,E1 28345.35,E2 28345.35} C_VEL
LIN {X 0,Y 591.918,Z 996.909,A -85,B 0,C 180,E1 28343.21,E2 28343.21} C_VEL
LIN {X 0,Y 591.931,Z 990.94,A -85,B 0,C 180,E1 28341.159,E2 28341.159} C_VEL
LIN {X 0,Y 591.947,Z 983.478,A -85,B 0,C 180,E1 28339.195,E2 28339.195} C_VEL
LIN {X 0,Y 591.991,Z 973.856,A -85,B 0,C 180,E1 28337.12,E2 28337.12} C_VEL
LIN {X 0,Y 592.058,Z 963.353,A -85,B 0,C 180,E1 28335.228,E2 28335.228} C_VEL
LIN {X 0,Y 592.132,Z 951.465,A -85,B 0,C 180,E1 28333.421,E2 28333.421} C_VEL
LIN {X 0,Y 592.243,Z 937.474,A -85,B 0,C 180,E1 28331.585,E2 28331.585} C_VEL
LIN {X 0,Y 592.393,Z 922.243,A -85,B 0,C 180,E1 28329.862,E2 28329.862} C_VEL
LIN {X 0,Y 592.564,Z 905.29,A -85,B 0,C 180,E1 28328.212,E2 28328.212} C_VEL
LIN {X 0,Y 592.72,Z 887.82,A -85,B 0,C 180,E1 28326.753,E2 28326.753} C_VEL
LIN {X 0,Y 592.934,Z 868.783,A -85,B 0,C 180,E1 28325.388,E2 28325.388} C_VEL
LIN {X 0,Y 593.151,Z 849.771,A -85,B 0,C 180,E1 28324.224,E2 28324.224} C_VEL
LIN {X 0,Y 593.294,Z 829.868,A -85,B 0,C 180,E1 28323.208,E2 28323.208} C_VEL
LIN {X 0,Y 593.507,Z 808.594,A -85,B 0,C 180,E1 28322.325,E2 28322.325} C_VEL
LIN {X 0,Y 593.681,Z 787.8,A -85,B 0,C 180,E1 28321.642,E2 28321.642} C_VEL
LIN {X 0,Y 593.763,Z 767.214,A -85,B 0,C 180,E1 28321.146,E2 28321.146} C_VEL
LIN {X 0,Y 593.881,Z 739.771,A -85,B 0,C 180,E1 28320.712,E2 28320.712} C_VEL
LIN {X 0,Y 594.27,Z 515.293,A -85,B 0,C 180,E1 28317.639,E2 28317.639} C_VEL
LIN {X 0,Y 594.222,Z 456.103,A -85,B 0,C 180,E1 28316.802,E2 28316.802} C_VEL
LIN {X 0,Y 593.984,Z 452.71,A -85,B 0,C 180,E1 28316.665,E2 28316.665} C_VEL
LIN {X 0,Y 594.396,Z 393.477,A -85,B 0,C 180,E1 28313.392,E2 28313.392} C_VEL
LIN {X 0,Y 594.555,Z 363.273,A -85,B 0,C 180,E1 28311.667,E2 28311.667} C_VEL
LIN {X 0,Y 592.081,Z 357.536,A -85,B 0,C 180,E1 28311.123,E2 28311.123} C_VEL
LIN {X 0,Y 592.009,Z 357.001,A -85,B 0,C 180,E1 28310.957,E2 28310.957} C_VEL
LIN {X 0,Y 591.978,Z 356.985,A -85,B 0,C 180,E1 28307.713,E2 28307.713} C_VEL
LIN {X 0,Y 592.003,Z 356.99,A -85,B 0,C 180,E1 28304.772,E2 28304.772} C_VEL
LIN {X 0,Y 591.976,Z 356.991,A -85,B 0,C 180,E1 28301.569,E2 28301.569} C_VEL
LIN {X 0,Y 591.989,Z 356.989,A -85,B 0,C 180,E1 28298.676,E2 28298.676} C_VEL
LIN {X 0,Y 591.972,Z 356.99,A -85,B 0,C 180,E1 28295.404,E2 28295.404} C_VEL
LIN {X 0,Y 591.978,Z 356.991,A -85,B 0,C 180,E1 28292.571,E2 28292.571} C_VEL
LIN {X 0,Y 591.974,Z 356.991,A -85,B 0,C 180,E1 28289.328,E2 28289.328} C_VEL
LIN {X 0,Y 591.967,Z 356.992,A -85,B 0,C 180,E1 28286.479,E2 28286.479} C_VEL
LIN {X 0,Y 591.963,Z 356.991,A -85,B 0,C 180,E1 28283.07,E2 28283.07} C_VEL
LIN {X 0,Y 591.964,Z 356.993,A -85,B 0,C 180,E1 28280.258,E2 28280.258} C_VEL
LIN {X 0,Y 591.956,Z 356.993,A -85,B 0,C 180,E1 28276.889,E2 28276.889} C_VEL
LIN {X 0,Y 591.955,Z 356.992,A -85,B 0,C 180,E1 28274.177,E2 28274.177} C_VEL
LIN {X 0,Y 591.975,Z 356.992,A -85,B 0,C 180,E1 28270.904,E2 28270.904} C_VEL
LIN {X 0,Y 591.956,Z 356.992,A -85,B 0,C 180,E1 28268.059,E2 28268.059} C_VEL
LIN {X 0,Y 591.992,Z 356.991,A -85,B 0,C 180,E1 28264.844,E2 28264.844} C_VEL
LIN {X 0,Y 591.96,Z 356.991,A -85,B 0,C 180,E1 28261.936,E2 28261.936} C_VEL
LIN {X 0,Y 592.007,Z 356.988,A -85,B 0,C 180,E1 28258.742,E2 28258.742} C_VEL
LIN {X 0,Y 591.963,Z 356.991,A -85,B 0,C 180,E1 28255.835,E2 28255.835} C_VEL
LIN {X 0,Y 592.032,Z 356.989,A -85,B 0,C 180,E1 28252.723,E2 28252.723} C_VEL
LIN {X 0,Y 591.972,Z 356.988,A -85,B 0,C 180,E1 28250.027,E2 28250.027} C_VEL
LIN {X 0,Y 590.973,Z 357.118,A -85,B 0,C 180,E1 28249.282,E2 28249.282} C_VEL
LIN {X 0,Y 584.624,Z 357.918,A -85,B 0,C 180,E1 28247.189,E2 28247.189} C_VEL
LIN {X 0,Y 584.1,Z 357.977,A -85,B 0,C 180,E1 28246.645,E2 28246.645} C_VEL
LIN {X 0,Y 584.033,Z 357.979,A -85,B 0,C 180,E1 28243.592,E2 28243.592} C_VEL
LIN {X 0,Y 584.101,Z 357.978,A -85,B 0,C 180,E1 28240.5,E2 28240.5} C_VEL
LIN {X 0,Y 584.04,Z 357.978,A -85,B 0,C 180,E1 28237.344,E2 28237.344} C_VEL
LIN {X 0,Y 584.093,Z 357.974,A -85,B 0,C 180,E1 28234.118,E2 28234.118} C_VEL
LIN {X 0,Y 584.048,Z 357.979,A -85,B 0,C 180,E1 28231.011,E2 28231.011} C_VEL
LIN {X 0,Y 584.077,Z 357.975,A -85,B 0,C 180,E1 28227.733,E2 28227.733} C_VEL
LIN {X 0,Y 584.075,Z 357.98,A -85,B 0,C 180,E1 28224.526,E2 28224.526} C_VEL
LIN {X 0,Y 584.054,Z 357.969,A -85,B 0,C 180,E1 28221.203,E2 28221.203} C_VEL
LIN {X 0,Y 584.094,Z 357.981,A -85,B 0,C 180,E1 28218.117,E2 28218.117} C_VEL
LIN {X 0,Y 584.055,Z 357.974,A -85,B 0,C 180,E1 28214.867,E2 28214.867} C_VEL
LIN {X 0,Y 584.095,Z 357.972,A -85,B 0,C 180,E1 28211.725,E2 28211.725} C_VEL
LIN {X 0,Y 584.059,Z 357.979,A -85,B 0,C 180,E1 28208.524,E2 28208.524} C_VEL
LIN {X 0,Y 584.095,Z 357.974,A -85,B 0,C 180,E1 28205.261,E2 28205.261} C_VEL
LIN {X 0,Y 584.075,Z 357.98,A -85,B 0,C 180,E1 28202.047,E2 28202.047} C_VEL
LIN {X 0,Y 584.121,Z 358.176,A -85,B 0,C 180,E1 28200.954,E2 28200.954} C_VEL
LIN {X 0,Y 585.951,Z 364.371,A -85,B 0,C 180,E1 28200.296,E2 28200.296} C_VEL
LIN {X 0,Y 585.868,Z 383.49,A -85,B 0,C 180,E1 28198.76,E2 28198.76} C_VEL
LIN {X 0,Y 586.707,Z 388.766,A -85,B 0,C 180,E1 28198.637,E2 28198.637} C_VEL
LIN {X 0,Y 586.074,Z 643.808,A -85,B 0,C 180,E1 28195.208,E2 28195.208} C_VEL
LIN {X 0,Y 585.919,Z 664.097,A -85,B 0,C 180,E1 28194.752,E2 28194.752} C_VEL
LIN {X 0,Y 585.733,Z 683.861,A -85,B 0,C 180,E1 28194.128,E2 28194.128} C_VEL
LIN {X 0,Y 585.504,Z 703.226,A -85,B 0,C 180,E1 28193.337,E2 28193.337} C_VEL
LIN {X 0,Y 585.299,Z 721.832,A -85,B 0,C 180,E1 28192.39,E2 28192.39} C_VEL
LIN {X 0,Y 585.056,Z 740.416,A -85,B 0,C 180,E1 28191.239,E2 28191.239} C_VEL
LIN {X 0,Y 584.803,Z 757.875,A -85,B 0,C 180,E1 28189.941,E2 28189.941} C_VEL
LIN {X 0,Y 584.581,Z 773.753,A -85,B 0,C 180,E1 28188.548,E2 28188.548} C_VEL
LIN {X 0,Y 584.389,Z 788.709,A -85,B 0,C 180,E1 28187.01,E2 28187.01} C_VEL
LIN {X 0,Y 584.233,Z 802.212,A -85,B 0,C 180,E1 28185.381,E2 28185.381} C_VEL
LIN {X 0,Y 584.102,Z 814.964,A -85,B 0,C 180,E1 28183.561,E2 28183.561} C_VEL
LIN {X 0,Y 584.017,Z 825.567,A -85,B 0,C 180,E1 28181.754,E2 28181.754} C_VEL
LIN {X 0,Y 583.962,Z 834.758,A -85,B 0,C 180,E1 28179.857,E2 28179.857} C_VEL
LIN {X 0,Y 583.936,Z 842.378,A -85,B 0,C 180,E1 28177.872,E2 28177.872} C_VEL
LIN {X 0,Y 583.923,Z 847.882,A -85,B 0,C 180,E1 28175.995,E2 28175.995} C_VEL
LIN {X 0,Y 583.918,Z 852.196,A -85,B 0,C 180,E1 28173.927,E2 28173.927} C_VEL
LIN {X 0,Y 583.916,Z 854.643,A -85,B 0,C 180,E1 28171.962,E2 28171.962} C_VEL
LIN {X 0,Y 583.914,Z 855.494,A -85,B 0,C 180,E1 28169.902,E2 28169.902} C_VEL
LIN {X 0,Y 583.913,Z 854.569,A -85,B 0,C 180,E1 28167.841,E2 28167.841} C_VEL
LIN {X 0,Y 583.917,Z 852.024,A -85,B 0,C 180,E1 28165.876,E2 28165.876} C_VEL
LIN {X 0,Y 583.925,Z 847.606,A -85,B 0,C 180,E1 28163.807,E2 28163.807} C_VEL
LIN {X 0,Y 583.942,Z 841.401,A -85,B 0,C 180,E1 28161.764,E2 28161.764} C_VEL
LIN {X 0,Y 583.971,Z 833.81,A -85,B 0,C 180,E1 28159.843,E2 28159.843} C_VEL
LIN {X 0,Y 584.037,Z 824.468,A -85,B 0,C 180,E1 28157.945,E2 28157.945} C_VEL
LIN {X 0,Y 584.125,Z 813.608,A -85,B 0,C 180,E1 28156.136,E2 28156.136} C_VEL
LIN {X 0,Y 584.24,Z 801.339,A -85,B 0,C 180,E1 28154.415,E2 28154.415} C_VEL
LIN {X 0,Y 584.394,Z 787.659,A -85,B 0,C 180,E1 28152.784,E2 28152.784} C_VEL
LIN {X 0,Y 584.597,Z 772.002,A -85,B 0,C 180,E1 28151.199,E2 28151.199} C_VEL
LIN {X 0,Y 584.826,Z 755.045,A -85,B 0,C 180,E1 28149.746,E2 28149.746} C_VEL
LIN {X 0,Y 585.081,Z 736.969,A -85,B 0,C 180,E1 28148.445,E2 28148.445} C_VEL
LIN {X 0,Y 585.331,Z 718.657,A -85,B 0,C 180,E1 28147.346,E2 28147.346} C_VEL
LIN {X 0,Y 585.583,Z 699.433,A -85,B 0,C 180,E1 28146.399,E2 28146.399} C_VEL
LIN {X 0,Y 585.773,Z 679.683,A -85,B 0,C 180,E1 28145.631,E2 28145.631} C_VEL
LIN {X 0,Y 585.94,Z 659.765,A -85,B 0,C 180,E1 28145.047,E2 28145.047} C_VEL
LIN {X 0,Y 586.087,Z 638.877,A -85,B 0,C 180,E1 28144.625,E2 28144.625} C_VEL
LIN {X 0,Y 586.71,Z 387.457,A -85,B 0,C 180,E1 28141.256,E2 28141.256} C_VEL
LIN {X 0,Y 585.79,Z 382.809,A -85,B 0,C 180,E1 28141.118,E2 28141.118} C_VEL
LIN {X 0,Y 585.803,Z 363.527,A -85,B 0,C 180,E1 28139.536,E2 28139.536} C_VEL
LIN {X 0,Y 584.127,Z 358.199,A -85,B 0,C 180,E1 28138.962,E2 28138.962} C_VEL
LIN {X 0,Y 584.072,Z 357.978,A -85,B 0,C 180,E1 28135.726,E2 28135.726} C_VEL
LIN {X 0,Y 584.093,Z 357.971,A -85,B 0,C 180,E1 28132.581,E2 28132.581} C_VEL
LIN {X 0,Y 584.063,Z 357.973,A -85,B 0,C 180,E1 28129.424,E2 28129.424} C_VEL
LIN {X 0,Y 584.094,Z 357.977,A -85,B 0,C 180,E1 28126.25,E2 28126.25} C_VEL
LIN {X 0,Y 584.058,Z 357.976,A -85,B 0,C 180,E1 28123.083,E2 28123.083} C_VEL
LIN {X 0,Y 584.1,Z 357.976,A -85,B 0,C 180,E1 28119.808,E2 28119.808} C_VEL
LIN {X 0,Y 584.067,Z 357.975,A -85,B 0,C 180,E1 28116.565,E2 28116.565} C_VEL
LIN {X 0,Y 584.062,Z 357.98,A -85,B 0,C 180,E1 28113.171,E2 28113.171} C_VEL
LIN {X 0,Y 584.103,Z 357.971,A -85,B 0,C 180,E1 28109.99,E2 28109.99} C_VEL
LIN {X 0,Y 584.048,Z 357.977,A -85,B 0,C 180,E1 28106.759,E2 28106.759} C_VEL
LIN {X 0,Y 584.099,Z 357.977,A -85,B 0,C 180,E1 28103.613,E2 28103.613} C_VEL
LIN {X 0,Y 584.042,Z 357.978,A -85,B 0,C 180,E1 28100.441,E2 28100.441} C_VEL
LIN {X 0,Y 584.099,Z 357.981,A -85,B 0,C 180,E1 28097.226,E2 28097.226} C_VEL
LIN {X 0,Y 584.038,Z 357.977,A -85,B 0,C 180,E1 28094.171,E2 28094.171} C_VEL
LIN {X 0,Y 584.084,Z 357.98,A -85,B 0,C 180,E1 28090.954,E2 28090.954} C_VEL
LIN {X 0,Y 584.037,Z 357.979,A -85,B 0,C 180,E1 28087.872,E2 28087.872} C_VEL
LIN {X 0,Y 584.059,Z 357.981,A -85,B 0,C 180,E1 28084.615,E2 28084.615} C_VEL
LIN {X 0,Y 584.032,Z 357.977,A -85,B 0,C 180,E1 28081.668,E2 28081.668} C_VEL
LIN {X 0,Y 584.043,Z 357.98,A -85,B 0,C 180,E1 28078.333,E2 28078.333} C_VEL
LIN {X 0,Y 584.034,Z 357.98,A -85,B 0,C 180,E1 28075.385,E2 28075.385} C_VEL
LIN {X 0,Y 584.027,Z 357.981,A -85,B 0,C 180,E1 28072.029,E2 28072.029} C_VEL
LIN {X 0,Y 584.024,Z 357.98,A -85,B 0,C 180,E1 28069.245,E2 28069.245} C_VEL
LIN {X 0,Y 584.027,Z 357.981,A -85,B 0,C 180,E1 28065.93,E2 28065.93} C_VEL
LIN {X 0,Y 584.018,Z 357.982,A -85,B 0,C 180,E1 28063.08,E2 28063.08} C_VEL
LIN {X 0,Y 584.024,Z 357.982,A -85,B 0,C 180,E1 28059.734,E2 28059.734} C_VEL
LIN {X 0,Y 584.022,Z 357.979,A -85,B 0,C 180,E1 28056.918,E2 28056.918} C_VEL
LIN {X 0,Y 584.029,Z 357.981,A -85,B 0,C 180,E1 28053.546,E2 28053.546} C_VEL
LIN {X 0,Y 584.031,Z 357.98,A -85,B 0,C 180,E1 28050.684,E2 28050.684} C_VEL
LIN {X 0,Y 584.033,Z 357.981,A -85,B 0,C 180,E1 28047.366,E2 28047.366} C_VEL
LIN {X 0,Y 584.036,Z 357.978,A -85,B 0,C 180,E1 28044.524,E2 28044.524} C_VEL
LIN {X 0,Y 584.037,Z 357.978,A -85,B 0,C 180,E1 28041.158,E2 28041.158} C_VEL
LIN {X 0,Y 584.051,Z 357.981,A -85,B 0,C 180,E1 28038.246,E2 28038.246} C_VEL
LIN {X 0,Y 584.044,Z 357.98,A -85,B 0,C 180,E1 28034.989,E2 28034.989} C_VEL
LIN {X 0,Y 584.061,Z 357.975,A -85,B 0,C 180,E1 28032.013,E2 28032.013} C_VEL
LIN {X 0,Y 584.11,Z 358.057,A -85,B 0,C 180,E1 28029.548,E2 28029.548} C_VEL
LIN {X 0,Y 584.434,Z 359.459,A -85,B 0,C 180,E1 28029.35,E2 28029.35} C_VEL
LIN {X 0,Y 587.984,Z 367.172,A -85,B 0,C 180,E1 28028.61,E2 28028.61} C_VEL
LIN {X 0,Y 587.387,Z 418.803,A -85,B 0,C 180,E1 28025.665,E2 28025.665} C_VEL
LIN {X 0,Y 587.175,Z 455.353,A -85,B 0,C 180,E1 28023.66,E2 28023.66} C_VEL
LIN {X 0,Y 587.701,Z 460.652,A -85,B 0,C 180,E1 28023.549,E2 28023.549} C_VEL
LIN {X 0,Y 587.041,Z 686.83,A -85,B 0,C 180,E1 28020.396,E2 28020.396} C_VEL
LIN {X 0,Y 586.801,Z 762.009,A -85,B 0,C 180,E1 28019.338,E2 28019.338} C_VEL
LIN {X 0,Y 586.614,Z 783.096,A -85,B 0,C 180,E1 28018.858,E2 28018.858} C_VEL
LIN {X 0,Y 586.369,Z 804.828,A -85,B 0,C 180,E1 28018.183,E2 28018.183} C_VEL
LIN {X 0,Y 586.144,Z 825.186,A -85,B 0,C 180,E1 28017.366,E2 28017.366} C_VEL
LIN {X 0,Y 585.831,Z 845.458,A -85,B 0,C 180,E1 28016.359,E2 28016.359} C_VEL
LIN {X 0,Y 585.521,Z 865.564,A -85,B 0,C 180,E1 28015.161,E2 28015.161} C_VEL
LIN {X 0,Y 585.248,Z 884.481,A -85,B 0,C 180,E1 28013.829,E2 28013.829} C_VEL
LIN {X 0,Y 584.944,Z 902.097,A -85,B 0,C 180,E1 28012.371,E2 28012.371} C_VEL
LIN {X 0,Y 584.675,Z 918.692,A -85,B 0,C 180,E1 28010.782,E2 28010.782} C_VEL
LIN {X 0,Y 584.471,Z 934.18,A -85,B 0,C 180,E1 28009.07,E2 28009.07} C_VEL
LIN {X 0,Y 584.299,Z 948.633,A -85,B 0,C 180,E1 28007.218,E2 28007.218} C_VEL
LIN {X 0,Y 584.155,Z 961.478,A -85,B 0,C 180,E1 28005.282,E2 28005.282} C_VEL
LIN {X 0,Y 584.047,Z 972.295,A -85,B 0,C 180,E1 28003.362,E2 28003.362} C_VEL
LIN {X 0,Y 583.981,Z 981.846,A -85,B 0,C 180,E1 28001.355,E2 28001.355} C_VEL
LIN {X 0,Y 583.931,Z 989.531,A -85,B 0,C 180,E1 27999.361,E2 27999.361} C_VEL
LIN {X 0,Y 583.903,Z 995.891,A -85,B 0,C 180,E1 27997.279,E2 27997.279} C_VEL
LIN {X 0,Y 583.9,Z 1000.427,A -85,B 0,C 180,E1 27995.305,E2 27995.305} C_VEL
LIN {X 0,Y 583.908,Z 1003.559,A -85,B 0,C 180,E1 27993.239,E2 27993.239} C_VEL
LIN {X 0,Y 583.913,Z 1005.262,A -85,B 0,C 180,E1 27991.08,E2 27991.08} C_VEL
LIN {X 0,Y 583.905,Z 1005.284,A -85,B 0,C 180,E1 27989.019,E2 27989.019} C_VEL
LIN {X 0,Y 583.902,Z 1003.672,A -85,B 0,C 180,E1 27986.86,E2 27986.86} C_VEL
LIN {X 0,Y 583.897,Z 1000.633,A -85,B 0,C 180,E1 27984.794,E2 27984.794} C_VEL
LIN {X 0,Y 583.904,Z 996.147,A -85,B 0,C 180,E1 27982.82,E2 27982.82} C_VEL
LIN {X 0,Y 583.934,Z 989.888,A -85,B 0,C 180,E1 27980.739,E2 27980.739} C_VEL
LIN {X 0,Y 583.98,Z 982.595,A -85,B 0,C 180,E1 27978.829,E2 27978.829} C_VEL
LIN {X 0,Y 584.044,Z 973.338,A -85,B 0,C 180,E1 27976.841,E2 27976.841} C_VEL
LIN {X 0,Y 584.152,Z 962.462,A -85,B 0,C 180,E1 27974.875,E2 27974.875} C_VEL
LIN {X 0,Y 584.276,Z 950.052,A -85,B 0,C 180,E1 27972.987,E2 27972.987} C_VEL
LIN {X 0,Y 584.444,Z 935.886,A -85,B 0,C 180,E1 27971.137,E2 27971.137} C_VEL
LIN {X 0,Y 584.662,Z 920.218,A -85,B 0,C 180,E1 27969.375,E2 27969.375} C_VEL
LIN {X 0,Y 584.927,Z 904.134,A -85,B 0,C 180,E1 27967.807,E2 27967.807} C_VEL
LIN {X 0,Y 585.202,Z 886.345,A -85,B 0,C 180,E1 27966.318,E2 27966.318} C_VEL
LIN {X 0,Y 585.472,Z 868.302,A -85,B 0,C 180,E1 27965.021,E2 27965.021} C_VEL
LIN {X 0,Y 585.806,Z 848.781,A -85,B 0,C 180,E1 27963.822,E2 27963.822} C_VEL
LIN {X 0,Y 586.039,Z 829.869,A -85,B 0,C 180,E1 27962.849,E2 27962.849} C_VEL
LIN {X 0,Y 586.338,Z 808.524,A -85,B 0,C 180,E1 27961.955,E2 27961.955} C_VEL
LIN {X 0,Y 586.6,Z 787.542,A -85,B 0,C 180,E1 27961.261,E2 27961.261} C_VEL
LIN {X 0,Y 586.735,Z 766.893,A -85,B 0,C 180,E1 27960.76,E2 27960.76} C_VEL
LIN {X 0,Y 586.905,Z 738.98,A -85,B 0,C 180,E1 27960.319,E2 27960.319} C_VEL
LIN {X 0,Y 587.513,Z 513.637,A -85,B 0,C 180,E1 27957.197,E2 27957.197} C_VEL
LIN {X 0,Y 587.512,Z 457.432,A -85,B 0,C 180,E1 27956.392,E2 27956.392} C_VEL
LIN {X 0,Y 587.058,Z 453.765,A -85,B 0,C 180,E1 27956.278,E2 27956.278} C_VEL
LIN {X 0,Y 587.679,Z 394.639,A -85,B 0,C 180,E1 27952.971,E2 27952.971} C_VEL
LIN {X 0,Y 587.898,Z 366.776,A -85,B 0,C 180,E1 27951.36,E2 27951.36} C_VEL
LIN {X 0,Y 584.181,Z 358.475,A -85,B 0,C 180,E1 27950.547,E2 27950.547} C_VEL
LIN {X 0,Y 584.089,Z 357.957,A -85,B 0,C 180,E1 27950.324,E2 27950.324} C_VEL
LIN {X 0,Y 584.033,Z 357.971,A -85,B 0,C 180,E1 27947.322,E2 27947.322} C_VEL
LIN {X 0,Y 584.093,Z 357.975,A -85,B 0,C 180,E1 27944.163,E2 27944.163} C_VEL
LIN {X 0,Y 584.03,Z 357.979,A -85,B 0,C 180,E1 27941.102,E2 27941.102} C_VEL
LIN {X 0,Y 584.077,Z 357.982,A -85,B 0,C 180,E1 27937.9,E2 27937.9} C_VEL
LIN {X 0,Y 584.026,Z 357.977,A -85,B 0,C 180,E1 27934.876,E2 27934.876} C_VEL
LIN {X 0,Y 584.07,Z 357.977,A -85,B 0,C 180,E1 27931.705,E2 27931.705} C_VEL
LIN {X 0,Y 584.02,Z 357.979,A -85,B 0,C 180,E1 27928.756,E2 27928.756} C_VEL
LIN {X 0,Y 584.068,Z 357.976,A -85,B 0,C 180,E1 27925.556,E2 27925.556} C_VEL
LIN {X 0,Y 584.013,Z 357.979,A -85,B 0,C 180,E1 27922.657,E2 27922.657} C_VEL
LIN {X 0,Y 584.081,Z 357.98,A -85,B 0,C 180,E1 27919.5,E2 27919.5} C_VEL
LIN {X 0,Y 584.007,Z 357.982,A -85,B 0,C 180,E1 27916.511,E2 27916.511} C_VEL
LIN {X 0,Y 584.086,Z 357.983,A -85,B 0,C 180,E1 27913.462,E2 27913.462} C_VEL
LIN {X 0,Y 584.01,Z 357.981,A -85,B 0,C 180,E1 27910.356,E2 27910.356} C_VEL
LIN {X 0,Y 584.098,Z 357.979,A -85,B 0,C 180,E1 27907.277,E2 27907.277} C_VEL
LIN {X 0,Y 584.017,Z 357.981,A -85,B 0,C 180,E1 27904.123,E2 27904.123} C_VEL
LIN {X 0,Y 584.09,Z 357.98,A -85,B 0,C 180,E1 27900.981,E2 27900.981} C_VEL
LIN {X 0,Y 584.022,Z 357.978,A -85,B 0,C 180,E1 27897.939,E2 27897.939} C_VEL
LIN {X 0,Y 584.092,Z 357.976,A -85,B 0,C 180,E1 27894.794,E2 27894.794} C_VEL
LIN {X 0,Y 584.027,Z 357.98,A -85,B 0,C 180,E1 27891.731,E2 27891.731} C_VEL
LIN {X 0,Y 584.09,Z 357.977,A -85,B 0,C 180,E1 27888.546,E2 27888.546} C_VEL
LIN {X 0,Y 584.1,Z 357.977,A -85,B 0,C 180,E1 27886.645,E2 27886.645} C_VEL
LIN {X 0,Y 583.096,Z 358.098,A -85,B 0,C 180,E1 27885.889,E2 27885.889} C_VEL
LIN {X 0,Y 576.616,Z 358.904,A -85,B 0,C 180,E1 27883.769,E2 27883.769} C_VEL
LIN {X 0,Y 576.108,Z 358.969,A -85,B 0,C 180,E1 27883.217,E2 27883.217} C_VEL
LIN {X 0,Y 576.11,Z 358.966,A -85,B 0,C 180,E1 27879.855,E2 27879.855} C_VEL
LIN {X 0,Y 576.134,Z 358.969,A -85,B 0,C 180,E1 27876.799,E2 27876.799} C_VEL
LIN {X 0,Y 576.106,Z 358.965,A -85,B 0,C 180,E1 27873.51,E2 27873.51} C_VEL
LIN {X 0,Y 576.162,Z 358.967,A -85,B 0,C 180,E1 27870.358,E2 27870.358} C_VEL
LIN {X 0,Y 576.107,Z 358.967,A -85,B 0,C 180,E1 27867.131,E2 27867.131} C_VEL
LIN {X 0,Y 576.16,Z 358.965,A -85,B 0,C 180,E1 27863.959,E2 27863.959} C_VEL
LIN {X 0,Y 576.112,Z 358.958,A -85,B 0,C 180,E1 27860.822,E2 27860.822} C_VEL
LIN {X 0,Y 576.156,Z 358.962,A -85,B 0,C 180,E1 27857.663,E2 27857.663} C_VEL
LIN {X 0,Y 576.122,Z 358.964,A -85,B 0,C 180,E1 27854.497,E2 27854.497} C_VEL
LIN {X 0,Y 576.136,Z 358.957,A -85,B 0,C 180,E1 27851.122,E2 27851.122} C_VEL
LIN {X 0,Y 576.157,Z 358.962,A -85,B 0,C 180,E1 27847.851,E2 27847.851} C_VEL
LIN {X 0,Y 576.123,Z 358.966,A -85,B 0,C 180,E1 27844.572,E2 27844.572} C_VEL
LIN {X 0,Y 576.18,Z 359.148,A -85,B 0,C 180,E1 27841.351,E2 27841.351} C_VEL
LIN {X 0,Y 578.636,Z 367.328,A -85,B 0,C 180,E1 27840.471,E2 27840.471} C_VEL
LIN {X 0,Y 578.527,Z 383.472,A -85,B 0,C 180,E1 27839.162,E2 27839.162} C_VEL
LIN {X 0,Y 579.681,Z 390.146,A -85,B 0,C 180,E1 27838.998,E2 27838.998} C_VEL
LIN {X 0,Y 578.833,Z 643.744,A -85,B 0,C 180,E1 27835.547,E2 27835.547} C_VEL
LIN {X 0,Y 578.628,Z 664.091,A -85,B 0,C 180,E1 27835.086,E2 27835.086} C_VEL
LIN {X 0,Y 578.374,Z 683.881,A -85,B 0,C 180,E1 27834.455,E2 27834.455} C_VEL
LIN {X 0,Y 578.085,Z 703.238,A -85,B 0,C 180,E1 27833.655,E2 27833.655} C_VEL
LIN {X 0,Y 577.794,Z 721.841,A -85,B 0,C 180,E1 27832.697,E2 27832.697} C_VEL
LIN {X 0,Y 577.462,Z 740.427,A -85,B 0,C 180,E1 27831.532,E2 27831.532} C_VEL
LIN {X 0,Y 577.123,Z 757.639,A -85,B 0,C 180,E1 27830.238,E2 27830.238} C_VEL
LIN {X 0,Y 576.824,Z 773.761,A -85,B 0,C 180,E1 27828.806,E2 27828.806} C_VEL
LIN {X 0,Y 576.564,Z 788.715,A -85,B 0,C 180,E1 27827.248,E2 27827.248} C_VEL
LIN {X 0,Y 576.353,Z 802.219,A -85,B 0,C 180,E1 27825.597,E2 27825.597} C_VEL
LIN {X 0,Y 576.183,Z 814.97,A -85,B 0,C 180,E1 27823.751,E2 27823.751} C_VEL
LIN {X 0,Y 576.065,Z 825.572,A -85,B 0,C 180,E1 27821.918,E2 27821.918} C_VEL
LIN {X 0,Y 575.984,Z 834.761,A -85,B 0,C 180,E1 27819.995,E2 27819.995} C_VEL
LIN {X 0,Y 575.945,Z 842.379,A -85,B 0,C 180,E1 27817.982,E2 27817.982} C_VEL
LIN {X 0,Y 575.926,Z 847.884,A -85,B 0,C 180,E1 27816.078,E2 27816.078} C_VEL
LIN {X 0,Y 575.918,Z 852.197,A -85,B 0,C 180,E1 27813.981,E2 27813.981} C_VEL
LIN {X 0,Y 575.916,Z 854.643,A -85,B 0,C 180,E1 27811.989,E2 27811.989} C_VEL
LIN {X 0,Y 575.914,Z 855.494,A -85,B 0,C 180,E1 27809.9,E2 27809.9} C_VEL
LIN {X 0,Y 575.911,Z 854.568,A -85,B 0,C 180,E1 27807.811,E2 27807.811} C_VEL
LIN {X 0,Y 575.918,Z 852.024,A -85,B 0,C 180,E1 27805.819,E2 27805.819} C_VEL
LIN {X 0,Y 575.927,Z 847.605,A -85,B 0,C 180,E1 27803.721,E2 27803.721} C_VEL
LIN {X 0,Y 575.952,Z 841.581,A -85,B 0,C 180,E1 27801.701,E2 27801.701} C_VEL
LIN {X 0,Y 575.993,Z 834.266,A -85,B 0,C 180,E1 27799.802,E2 27799.802} C_VEL
LIN {X 0,Y 576.078,Z 824.988,A -85,B 0,C 180,E1 27797.878,E2 27797.878} C_VEL
LIN {X 0,Y 576.196,Z 814.245,A -85,B 0,C 180,E1 27796.044,E2 27796.044} C_VEL
LIN {X 0,Y 576.354,Z 802.111,A -85,B 0,C 180,E1 27794.3,E2 27794.3} C_VEL
LIN {X 0,Y 576.564,Z 788.58,A -85,B 0,C 180,E1 27792.647,E2 27792.647} C_VEL
LIN {X 0,Y 576.826,Z 773.599,A -85,B 0,C 180,E1 27791.088,E2 27791.088} C_VEL
LIN {X 0,Y 577.125,Z 757.683,A -85,B 0,C 180,E1 27789.676,E2 27789.676} C_VEL
LIN {X 0,Y 577.465,Z 740.171,A -85,B 0,C 180,E1 27788.36,E2 27788.36} C_VEL
LIN {X 0,Y 577.797,Z 721.53,A -85,B 0,C 180,E1 27787.195,E2 27787.195} C_VEL
LIN {X 0,Y 578.094,Z 702.846,A -85,B 0,C 180,E1 27786.237,E2 27786.237} C_VEL
LIN {X 0,Y 578.371,Z 683.757,A -85,B 0,C 180,E1 27785.45,E2 27785.45} C_VEL
LIN {X 0,Y 578.634,Z 663.248,A -85,B 0,C 180,E1 27784.802,E2 27784.802} C_VEL
LIN {X 0,Y 578.837,Z 643.026,A -85,B 0,C 180,E1 27784.352,E2 27784.352} C_VEL
LIN {X 0,Y 579.688,Z 389.03,A -85,B 0,C 180,E1 27780.897,E2 27780.897} C_VEL
LIN {X 0,Y 578.455,Z 382.817,A -85,B 0,C 180,E1 27780.717,E2 27780.717} C_VEL
LIN {X 0,Y 578.467,Z 366.341,A -85,B 0,C 180,E1 27779.346,E2 27779.346} C_VEL
LIN {X 0,Y 576.189,Z 359.231,A -85,B 0,C 180,E1 27778.579,E2 27778.579} C_VEL
LIN {X 0,Y 576.155,Z 358.967,A -85,B 0,C 180,E1 27776.951,E2 27776.951} C_VEL
LIN {X 0,Y 576.129,Z 358.964,A -85,B 0,C 180,E1 27773.596,E2 27773.596} C_VEL
LIN {X 0,Y 576.154,Z 358.966,A -85,B 0,C 180,E1 27770.401,E2 27770.401} C_VEL
LIN {X 0,Y 576.122,Z 358.967,A -85,B 0,C 180,E1 27767.233,E2 27767.233} C_VEL
LIN {X 0,Y 576.157,Z 358.961,A -85,B 0,C 180,E1 27763.96,E2 27763.96} C_VEL
LIN {X 0,Y 576.132,Z 358.964,A -85,B 0,C 180,E1 27760.683,E2 27760.683} C_VEL
LIN {X 0,Y 576.125,Z 358.968,A -85,B 0,C 180,E1 27757.278,E2 27757.278} C_VEL
LIN {X 0,Y 576.16,Z 358.962,A -85,B 0,C 180,E1 27754.093,E2 27754.093} C_VEL
LIN {X 0,Y 576.112,Z 358.965,A -85,B 0,C 180,E1 27750.912,E2 27750.912} C_VEL
LIN {X 0,Y 576.162,Z 358.966,A -85,B 0,C 180,E1 27747.716,E2 27747.716} C_VEL
LIN {X 0,Y 576.106,Z 358.966,A -85,B 0,C 180,E1 27744.507,E2 27744.507} C_VEL
LIN {X 0,Y 576.154,Z 358.971,A -85,B 0,C 180,E1 27741.266,E2 27741.266} C_VEL
LIN {X 0,Y 576.111,Z 358.965,A -85,B 0,C 180,E1 27738.099,E2 27738.099} C_VEL
LIN {X 0,Y 576.11,Z 358.968,A -85,B 0,C 180,E1 27734.678,E2 27734.678} C_VEL
LIN {X 0,Y 576.131,Z 358.966,A -85,B 0,C 180,E1 27731.614,E2 27731.614} C_VEL
LIN {X 0,Y 576.099,Z 358.969,A -85,B 0,C 180,E1 27728.383,E2 27728.383} C_VEL
LIN {X 0,Y 576.144,Z 358.963,A -85,B 0,C 180,E1 27725.278,E2 27725.278} C_VEL
LIN {X 0,Y 576.088,Z 358.966,A -85,B 0,C 180,E1 27722.089,E2 27722.089} C_VEL
LIN {X 0,Y 576.153,Z 358.968,A -85,B 0,C 180,E1 27719.006,E2 27719.006} C_VEL
LIN {X 0,Y 576.081,Z 358.97,A -85,B 0,C 180,E1 27715.82,E2 27715.82} C_VEL
LIN {X 0,Y 576.159,Z 358.967,A -85,B 0,C 180,E1 27712.722,E2 27712.722} C_VEL
LIN {X 0,Y 576.074,Z 358.969,A -85,B 0,C 180,E1 27709.601,E2 27709.601} C_VEL
LIN {X 0,Y 576.149,Z 358.971,A -85,B 0,C 180,E1 27706.451,E2 27706.451} C_VEL
LIN {X 0,Y 576.069,Z 358.971,A -85,B 0,C 180,E1 27703.359,E2 27703.359} C_VEL
LIN {X 0,Y 576.137,Z 358.972,A -85,B 0,C 180,E1 27700.22,E2 27700.22} C_VEL
LIN {X 0,Y 576.074,Z 358.968,A -85,B 0,C 180,E1 27697.121,E2 27697.121} C_VEL
LIN {X 0,Y 576.132,Z 358.97,A -85,B 0,C 180,E1 27693.956,E2 27693.956} C_VEL
LIN {X 0,Y 576.08,Z 358.969,A -85,B 0,C 180,E1 27690.924,E2 27690.924} C_VEL
LIN {X 0,Y 576.142,Z 358.969,A -85,B 0,C 180,E1 27687.807,E2 27687.807} C_VEL
LIN {X 0,Y 576.085,Z 358.965,A -85,B 0,C 180,E1 27684.815,E2 27684.815} C_VEL
LIN {X 0,Y 576.142,Z 358.966,A -85,B 0,C 180,E1 27681.59,E2 27681.59} C_VEL
LIN {X 0,Y 576.093,Z 358.969,A -85,B 0,C 180,E1 27678.565,E2 27678.565} C_VEL
LIN {X 0,Y 576.138,Z 358.967,A -85,B 0,C 180,E1 27675.344,E2 27675.344} C_VEL
LIN {X 0,Y 576.099,Z 358.962,A -85,B 0,C 180,E1 27672.324,E2 27672.324} C_VEL
LIN {X 0,Y 576.124,Z 359.083,A -85,B 0,C 180,E1 27670.141,E2 27670.141} C_VEL
LIN {X 0,Y 576.446,Z 360.415,A -85,B 0,C 180,E1 27669.946,E2 27669.946} C_VEL
LIN {X 0,Y 581.361,Z 370.567,A -85,B 0,C 180,E1 27668.93,E2 27668.93} C_VEL
LIN {X 0,Y 580.596,Z 421.125,A -85,B 0,C 180,E1 27666.013,E2 27666.013} C_VEL
LIN {X 0,Y 580.28,Z 455.281,A -85,B 0,C 180,E1 27664.116,E2 27664.116} C_VEL
LIN {X 0,Y 581.026,Z 461.704,A -85,B 0,C 180,E1 27663.972,E2 27663.972} C_VEL
LIN {X 0,Y 580.135,Z 688.102,A -85,B 0,C 180,E1 27660.779,E2 27660.779} C_VEL
LIN {X 0,Y 579.819,Z 762.116,A -85,B 0,C 180,E1 27659.725,E2 27659.725} C_VEL
LIN {X 0,Y 579.565,Z 783.356,A -85,B 0,C 180,E1 27659.236,E2 27659.236} C_VEL
LIN {X 0,Y 579.252,Z 804.824,A -85,B 0,C 180,E1 27658.561,E2 27658.561} C_VEL
LIN {X 0,Y 578.937,Z 825.189,A -85,B 0,C 180,E1 27657.736,E2 27657.736} C_VEL
LIN {X 0,Y 578.525,Z 844.792,A -85,B 0,C 180,E1 27656.755,E2 27656.755} C_VEL
LIN {X 0,Y 578.136,Z 864.753,A -85,B 0,C 180,E1 27655.56,E2 27655.56} C_VEL
LIN {X 0,Y 577.736,Z 883.814,A -85,B 0,C 180,E1 27654.21,E2 27654.21} C_VEL
LIN {X 0,Y 577.325,Z 901.713,A -85,B 0,C 180,E1 27652.717,E2 27652.717} C_VEL
LIN {X 0,Y 576.966,Z 918.825,A -85,B 0,C 180,E1 27651.059,E2 27651.059} C_VEL
LIN {X 0,Y 576.682,Z 934.181,A -85,B 0,C 180,E1 27649.337,E2 27649.337} C_VEL
LIN {X 0,Y 576.437,Z 948.634,A -85,B 0,C 180,E1 27647.461,E2 27647.461} C_VEL
LIN {X 0,Y 576.237,Z 960.838,A -85,B 0,C 180,E1 27645.6,E2 27645.6} C_VEL
LIN {X 0,Y 576.093,Z 972.297,A -85,B 0,C 180,E1 27643.55,E2 27643.55} C_VEL
LIN {X 0,Y 576.005,Z 981.847,A -85,B 0,C 180,E1 27641.514,E2 27641.514} C_VEL
LIN {X 0,Y 575.943,Z 989.235,A -85,B 0,C 180,E1 27639.577,E2 27639.577} C_VEL
LIN {X 0,Y 575.908,Z 995.891,A -85,B 0,C 180,E1 27637.381,E2 27637.381} C_VEL
LIN {X 0,Y 575.905,Z 1000.427,A -85,B 0,C 180,E1 27635.379,E2 27635.379} C_VEL
LIN {X 0,Y 575.912,Z 1003.56,A -85,B 0,C 180,E1 27633.284,E2 27633.284} C_VEL
LIN {X 0,Y 575.913,Z 1005.262,A -85,B 0,C 180,E1 27631.095,E2 27631.095} C_VEL
LIN {X 0,Y 575.907,Z 1005.284,A -85,B 0,C 180,E1 27629.006,E2 27629.006} C_VEL
LIN {X 0,Y 575.904,Z 1003.672,A -85,B 0,C 180,E1 27626.816,E2 27626.816} C_VEL
LIN {X 0,Y 575.9,Z 1000.633,A -85,B 0,C 180,E1 27624.721,E2 27624.721} C_VEL
LIN {X 0,Y 575.907,Z 996.147,A -85,B 0,C 180,E1 27622.72,E2 27622.72} C_VEL
LIN {X 0,Y 575.944,Z 989.889,A -85,B 0,C 180,E1 27620.609,E2 27620.609} C_VEL
LIN {X 0,Y 576.003,Z 982.664,A -85,B 0,C 180,E1 27618.689,E2 27618.689} C_VEL
LIN {X 0,Y 576.093,Z 973.339,A -85,B 0,C 180,E1 27616.656,E2 27616.656} C_VEL
LIN {X 0,Y 576.234,Z 962.751,A -85,B 0,C 180,E1 27614.71,E2 27614.71} C_VEL
LIN {X 0,Y 576.399,Z 950.76,A -85,B 0,C 180,E1 27612.851,E2 27612.851} C_VEL
LIN {X 0,Y 576.63,Z 936.737,A -85,B 0,C 180,E1 27610.977,E2 27610.977} C_VEL
LIN {X 0,Y 576.919,Z 921.658,A -85,B 0,C 180,E1 27609.237,E2 27609.237} C_VEL
LIN {X 0,Y 577.283,Z 904.759,A -85,B 0,C 180,E1 27607.554,E2 27607.554} C_VEL
LIN {X 0,Y 577.669,Z 886.492,A -85,B 0,C 180,E1 27606.002,E2 27606.002} C_VEL
LIN {X 0,Y 578.042,Z 867.986,A -85,B 0,C 180,E1 27604.656,E2 27604.656} C_VEL
LIN {X 0,Y 578.476,Z 848.783,A -85,B 0,C 180,E1 27603.465,E2 27603.465} C_VEL
LIN {X 0,Y 578.817,Z 829.866,A -85,B 0,C 180,E1 27602.482,E2 27602.482} C_VEL
LIN {X 0,Y 579.195,Z 808.527,A -85,B 0,C 180,E1 27601.577,E2 27601.577} C_VEL
LIN {X 0,Y 579.545,Z 787.414,A -85,B 0,C 180,E1 27600.874,E2 27600.874} C_VEL
LIN {X 0,Y 579.736,Z 766.498,A -85,B 0,C 180,E1 27600.364,E2 27600.364} C_VEL
LIN {X 0,Y 579.959,Z 737.765,A -85,B 0,C 180,E1 27599.91,E2 27599.91} C_VEL
LIN {X 0,Y 580.794,Z 511.444,A -85,B 0,C 180,E1 27596.737,E2 27596.737} C_VEL
LIN {X 0,Y 580.835,Z 458.757,A -85,B 0,C 180,E1 27595.973,E2 27595.973} C_VEL
LIN {X 0,Y 580.178,Z 453.598,A -85,B 0,C 180,E1 27595.813,E2 27595.813} C_VEL
LIN {X 0,Y 581.013,Z 394.639,A -85,B 0,C 180,E1 27592.474,E2 27592.474} C_VEL
LIN {X 0,Y 581.195,Z 370.294,A -85,B 0,C 180,E1 27591.041,E2 27591.041} C_VEL
LIN {X 0,Y 577.396,Z 362.346,A -85,B 0,C 180,E1 27590.251,E2 27590.251} C_VEL
LIN {X 0,Y 576.173,Z 359.352,A -85,B 0,C 180,E1 27589.929,E2 27589.929} C_VEL
LIN {X 0,Y 576.096,Z 358.962,A -85,B 0,C 180,E1 27589.48,E2 27589.48} C_VEL
LIN {X 0,Y 576.16,Z 358.963,A -85,B 0,C 180,E1 27586.322,E2 27586.322} C_VEL
LIN {X 0,Y 576.092,Z 358.968,A -85,B 0,C 180,E1 27583.208,E2 27583.208} C_VEL
LIN {X 0,Y 576.139,Z 358.964,A -85,B 0,C 180,E1 27579.949,E2 27579.949} C_VEL
LIN {X 0,Y 576.091,Z 358.968,A -85,B 0,C 180,E1 27576.906,E2 27576.906} C_VEL
LIN {X 0,Y 576.113,Z 358.971,A -85,B 0,C 180,E1 27573.596,E2 27573.596} C_VEL
LIN {X 0,Y 576.088,Z 358.963,A -85,B 0,C 180,E1 27570.681,E2 27570.681} C_VEL
LIN {X 0,Y 576.104,Z 358.971,A -85,B 0,C 180,E1 27567.382,E2 27567.382} C_VEL
LIN {X 0,Y 576.08,Z 358.963,A -85,B 0,C 180,E1 27564.507,E2 27564.507} C_VEL
LIN {X 0,Y 576.105,Z 358.971,A -85,B 0,C 180,E1 27561.268,E2 27561.268} C_VEL
LIN {X 0,Y 576.078,Z 358.969,A -85,B 0,C 180,E1 27558.309,E2 27558.309} C_VEL
LIN {X 0,Y 576.09,Z 358.97,A -85,B 0,C 180,E1 27554.987,E2 27554.987} C_VEL
LIN {X 0,Y 576.078,Z 358.971,A -85,B 0,C 180,E1 27552.123,E2 27552.123} C_VEL
LIN {X 0,Y 576.093,Z 358.97,A -85,B 0,C 180,E1 27548.785,E2 27548.785} C_VEL
LIN {X 0,Y 576.082,Z 358.969,A -85,B 0,C 180,E1 27545.977,E2 27545.977} C_VEL
LIN {X 0,Y 576.106,Z 358.967,A -85,B 0,C 180,E1 27542.686,E2 27542.686} C_VEL
LIN {X 0,Y 576.088,Z 358.97,A -85,B 0,C 180,E1 27539.801,E2 27539.801} C_VEL
LIN {X 0,Y 576.112,Z 358.968,A -85,B 0,C 180,E1 27536.517,E2 27536.517} C_VEL
LIN {X 0,Y 576.099,Z 358.966,A -85,B 0,C 180,E1 27533.522,E2 27533.522} C_VEL
LIN {X 0,Y 576.099,Z 358.965,A -85,B 0,C 180,E1 27530.106,E2 27530.106} C_VEL
LIN {X 0,Y 576.119,Z 358.97,A -85,B 0,C 180,E1 27527.165,E2 27527.165} C_VEL
LIN {X 0,Y 576.101,Z 358.967,A -85,B 0,C 180,E1 27523.877,E2 27523.877} C_VEL
LIN {X 0,Y 576.108,Z 358.969,A -85,B 0,C 180,E1 27523.217,E2 27523.217} C_VEL
LIN {X 0,Y 575.158,Z 359.094,A -85,B 0,C 180,E1 27522.451,E2 27522.451} C_VEL
LIN {X 0,Y 568.62,Z 359.903,A -85,B 0,C 180,E1 27520.245,E2 27520.245} C_VEL
LIN {X 0,Y 568.165,Z 359.956,A -85,B 0,C 180,E1 27519.74,E2 27519.74} C_VEL
LIN {X 0,Y 568.218,Z 359.956,A -85,B 0,C 180,E1 27516.567,E2 27516.567} C_VEL
LIN {X 0,Y 568.164,Z 359.955,A -85,B 0,C 180,E1 27513.336,E2 27513.336} C_VEL
LIN {X 0,Y 568.223,Z 359.952,A -85,B 0,C 180,E1 27510.134,E2 27510.134} C_VEL
LIN {X 0,Y 568.172,Z 359.958,A -85,B 0,C 180,E1 27506.939,E2 27506.939} C_VEL
LIN {X 0,Y 568.202,Z 359.952,A -85,B 0,C 180,E1 27503.629,E2 27503.629} C_VEL
LIN {X 0,Y 568.199,Z 359.947,A -85,B 0,C 180,E1 27500.414,E2 27500.414} C_VEL
LIN {X 0,Y 568.18,Z 359.953,A -85,B 0,C 180,E1 27497.053,E2 27497.053} C_VEL
LIN {X 0,Y 568.22,Z 359.957,A -85,B 0,C 180,E1 27493.825,E2 27493.825} C_VEL
LIN {X 0,Y 568.18,Z 359.948,A -85,B 0,C 180,E1 27490.62,E2 27490.62} C_VEL
LIN {X 0,Y 568.216,Z 359.945,A -85,B 0,C 180,E1 27487.374,E2 27487.374} C_VEL
LIN {X 0,Y 568.194,Z 359.951,A -85,B 0,C 180,E1 27484.145,E2 27484.145} C_VEL
LIN {X 0,Y 568.251,Z 360.201,A -85,B 0,C 180,E1 27481.738,E2 27481.738} C_VEL
LIN {X 0,Y 571.33,Z 370.059,A -85,B 0,C 180,E1 27480.669,E2 27480.669} C_VEL
LIN {X 0,Y 571.209,Z 383.43,A -85,B 0,C 180,E1 27479.575,E2 27479.575} C_VEL
LIN {X 0,Y 572.68,Z 391.563,A -85,B 0,C 180,E1 27479.368,E2 27479.368} C_VEL
LIN {X 0,Y 571.613,Z 643.572,A -85,B 0,C 180,E1 27475.897,E2 27475.897} C_VEL
LIN {X 0,Y 571.359,Z 663.938,A -85,B 0,C 180,E1 27475.432,E2 27475.432} C_VEL
LIN {X 0,Y 571.035,Z 683.902,A -85,B 0,C 180,E1 27474.791,E2 27474.791} C_VEL
LIN {X 0,Y 570.661,Z 704.053,A -85,B 0,C 180,E1 27473.942,E2 27473.942} C_VEL
LIN {X 0,Y 570.282,Z 722.659,A -85,B 0,C 180,E1 27472.964,E2 27472.964} C_VEL
LIN {X 0,Y 569.881,Z 740.437,A -85,B 0,C 180,E1 27471.834,E2 27471.834} C_VEL
LIN {X 0,Y 569.452,Z 757.897,A -85,B 0,C 180,E1 27470.502,E2 27470.502} C_VEL
LIN {X 0,Y 569.076,Z 774.05,A -85,B 0,C 180,E1 27469.045,E2 27469.045} C_VEL
LIN {X 0,Y 568.754,Z 788.721,A -85,B 0,C 180,E1 27467.492,E2 27467.492} C_VEL
LIN {X 0,Y 568.483,Z 802.226,A -85,B 0,C 180,E1 27465.818,E2 27465.818} C_VEL
LIN {X 0,Y 568.266,Z 814.975,A -85,B 0,C 180,E1 27463.947,E2 27463.947} C_VEL
LIN {X 0,Y 568.116,Z 825.577,A -85,B 0,C 180,E1 27462.088,E2 27462.088} C_VEL
LIN {X 0,Y 568.01,Z 834.764,A -85,B 0,C 180,E1 27460.137,E2 27460.137} C_VEL
LIN {X 0,Y 567.955,Z 842.381,A -85,B 0,C 180,E1 27458.095,E2 27458.095} C_VEL
LIN {X 0,Y 567.93,Z 847.885,A -85,B 0,C 180,E1 27456.164,E2 27456.164} C_VEL
LIN {X 0,Y 567.919,Z 852.199,A -85,B 0,C 180,E1 27454.038,E2 27454.038} C_VEL
LIN {X 0,Y 567.916,Z 854.643,A -85,B 0,C 180,E1 27452.017,E2 27452.017} C_VEL
LIN {X 0,Y 567.914,Z 855.494,A -85,B 0,C 180,E1 27449.899,E2 27449.899} C_VEL
LIN {X 0,Y 567.91,Z 854.567,A -85,B 0,C 180,E1 27447.78,E2 27447.78} C_VEL
LIN {X 0,Y 567.916,Z 852.024,A -85,B 0,C 180,E1 27445.76,E2 27445.76} C_VEL
LIN {X 0,Y 567.93,Z 847.857,A -85,B 0,C 180,E1 27443.734,E2 27443.734} C_VEL
LIN {X 0,Y 567.961,Z 841.985,A -85,B 0,C 180,E1 27441.701,E2 27441.701} C_VEL
LIN {X 0,Y 568.017,Z 834.597,A -85,B 0,C 180,E1 27439.733,E2 27439.733} C_VEL
LIN {X 0,Y 568.119,Z 825.504,A -85,B 0,C 180,E1 27437.809,E2 27437.809} C_VEL
LIN {X 0,Y 568.267,Z 814.881,A -85,B 0,C 180,E1 27435.949,E2 27435.949} C_VEL
LIN {X 0,Y 568.471,Z 802.837,A -85,B 0,C 180,E1 27434.175,E2 27434.175} C_VEL
LIN {X 0,Y 568.735,Z 789.501,A -85,B 0,C 180,E1 27432.506,E2 27432.506} C_VEL
LIN {X 0,Y 569.065,Z 774.698,A -85,B 0,C 180,E1 27430.927,E2 27430.927} C_VEL
LIN {X 0,Y 569.449,Z 758.339,A -85,B 0,C 180,E1 27429.443,E2 27429.443} C_VEL
LIN {X 0,Y 569.868,Z 740.915,A -85,B 0,C 180,E1 27428.111,E2 27428.111} C_VEL
LIN {X 0,Y 570.286,Z 722.338,A -85,B 0,C 180,E1 27426.927,E2 27426.927} C_VEL
LIN {X 0,Y 570.664,Z 703.961,A -85,B 0,C 180,E1 27425.963,E2 27425.963} C_VEL
LIN {X 0,Y 571.03,Z 684.001,A -85,B 0,C 180,E1 27425.122,E2 27425.122} C_VEL
LIN {X 0,Y 571.361,Z 663.744,A -85,B 0,C 180,E1 27424.472,E2 27424.472} C_VEL
LIN {X 0,Y 571.615,Z 643.52,A -85,B 0,C 180,E1 27424.012,E2 27424.012} C_VEL
LIN {X 0,Y 572.679,Z 392.163,A -85,B 0,C 180,E1 27420.551,E2 27420.551} C_VEL
LIN {X 0,Y 572.19,Z 388.076,A -85,B 0,C 180,E1 27420.465,E2 27420.465} C_VEL
LIN {X 0,Y 571.143,Z 382.821,A -85,B 0,C 180,E1 27420.305,E2 27420.305} C_VEL
LIN {X 0,Y 571.264,Z 369.524,A -85,B 0,C 180,E1 27419.191,E2 27419.191} C_VEL
LIN {X 0,Y 568.269,Z 360.316,A -85,B 0,C 180,E1 27418.193,E2 27418.193} C_VEL
LIN {X 0,Y 568.193,Z 359.958,A -85,B 0,C 180,E1 27417.636,E2 27417.636} C_VEL
LIN {X 0,Y 568.215,Z 359.957,A -85,B 0,C 180,E1 27414.381,E2 27414.381} C_VEL
LIN {X 0,Y 568.195,Z 359.955,A -85,B 0,C 180,E1 27411.059,E2 27411.059} C_VEL
LIN {X 0,Y 568.198,Z 359.959,A -85,B 0,C 180,E1 27407.631,E2 27407.631} C_VEL
LIN {X 0,Y 568.218,Z 359.947,A -85,B 0,C 180,E1 27404.313,E2 27404.313} C_VEL
LIN {X 0,Y 568.181,Z 359.955,A -85,B 0,C 180,E1 27401.025,E2 27401.025} C_VEL
LIN {X 0,Y 568.219,Z 359.947,A -85,B 0,C 180,E1 27397.76,E2 27397.76} C_VEL
LIN {X 0,Y 568.186,Z 359.953,A -85,B 0,C 180,E1 27394.516,E2 27394.516} C_VEL
LIN {X 0,Y 568.184,Z 359.955,A -85,B 0,C 180,E1 27391.156,E2 27391.156} C_VEL
LIN {X 0,Y 568.221,Z 359.953,A -85,B 0,C 180,E1 27387.909,E2 27387.909} C_VEL
LIN {X 0,Y 568.167,Z 359.956,A -85,B 0,C 180,E1 27384.65,E2 27384.65} C_VEL
LIN {X 0,Y 568.223,Z 359.956,A -85,B 0,C 180,E1 27381.448,E2 27381.448} C_VEL
LIN {X 0,Y 568.165,Z 359.954,A -85,B 0,C 180,E1 27378.255,E2 27378.255} C_VEL
LIN {X 0,Y 568.199,Z 359.957,A -85,B 0,C 180,E1 27374.988,E2 27374.988} C_VEL
LIN {X 0,Y 568.169,Z 359.956,A -85,B 0,C 180,E1 27371.882,E2 27371.882} C_VEL
LIN {X 0,Y 568.165,Z 359.959,A -85,B 0,C 180,E1 27368.501,E2 27368.501} C_VEL
LIN {X 0,Y 568.186,Z 359.952,A -85,B 0,C 180,E1 27365.453,E2 27365.453} C_VEL
LIN {X 0,Y 568.154,Z 359.955,A -85,B 0,C 180,E1 27362.219,E2 27362.219} C_VEL
LIN {X 0,Y 568.19,Z 359.957,A -85,B 0,C 180,E1 27359.194,E2 27359.194} C_VEL
LIN {X 0,Y 568.145,Z 359.959,A -85,B 0,C 180,E1 27355.964,E2 27355.964} C_VEL
LIN {X 0,Y 568.209,Z 359.956,A -85,B 0,C 180,E1 27352.823,E2 27352.823} C_VEL
LIN {X 0,Y 568.136,Z 359.958,A -85,B 0,C 180,E1 27349.637,E2 27349.637} C_VEL
LIN {X 0,Y 568.21,Z 359.96,A -85,B 0,C 180,E1 27346.466,E2 27346.466} C_VEL
LIN {X 0,Y 568.131,Z 359.96,A -85,B 0,C 180,E1 27343.435,E2 27343.435} C_VEL
LIN {X 0,Y 568.201,Z 359.961,A -85,B 0,C 180,E1 27340.254,E2 27340.254} C_VEL
LIN {X 0,Y 568.135,Z 359.956,A -85,B 0,C 180,E1 27337.112,E2 27337.112} C_VEL
LIN {X 0,Y 568.185,Z 359.96,A -85,B 0,C 180,E1 27333.901,E2 27333.901} C_VEL
LIN {X 0,Y 568.141,Z 359.958,A -85,B 0,C 180,E1 27330.94,E2 27330.94} C_VEL
LIN {X 0,Y 568.199,Z 359.959,A -85,B 0,C 180,E1 27327.779,E2 27327.779} C_VEL
LIN {X 0,Y 568.149,Z 359.954,A -85,B 0,C 180,E1 27324.735,E2 27324.735} C_VEL
LIN {X 0,Y 568.187,Z 359.956,A -85,B 0,C 180,E1 27321.469,E2 27321.469} C_VEL
LIN {X 0,Y 568.159,Z 359.958,A -85,B 0,C 180,E1 27318.437,E2 27318.437} C_VEL
LIN {X 0,Y 568.169,Z 359.96,A -85,B 0,C 180,E1 27315.021,E2 27315.021} C_VEL
LIN {X 0,Y 568.188,Z 359.949,A -85,B 0,C 180,E1 27311.962,E2 27311.962} C_VEL
LIN {X 0,Y 568.193,Z 360.181,A -85,B 0,C 180,E1 27310.719,E2 27310.719} C_VEL
LIN {X 0,Y 569.163,Z 362.949,A -85,B 0,C 180,E1 27310.404,E2 27310.404} C_VEL
LIN {X 0,Y 572.385,Z 369.284,A -85,B 0,C 180,E1 27309.738,E2 27309.738} C_VEL
LIN {X 0,Y 574.765,Z 374.936,A -85,B 0,C 180,E1 27309.196,E2 27309.196} C_VEL
LIN {X 0,Y 573.773,Z 426.299,A -85,B 0,C 180,E1 27306.206,E2 27306.206} C_VEL
LIN {X 0,Y 573.436,Z 455.288,A -85,B 0,C 180,E1 27304.582,E2 27304.582} C_VEL
LIN {X 0,Y 574.382,Z 462.886,A -85,B 0,C 180,E1 27304.402,E2 27304.402} C_VEL
LIN {X 0,Y 573.255,Z 689.375,A -85,B 0,C 180,E1 27301.171,E2 27301.171} C_VEL
LIN {X 0,Y 572.864,Z 762.219,A -85,B 0,C 180,E1 27300.121,E2 27300.121} C_VEL
LIN {X 0,Y 572.541,Z 783.616,A -85,B 0,C 180,E1 27299.622,E2 27299.622} C_VEL
LIN {X 0,Y 572.142,Z 805.626,A -85,B 0,C 180,E1 27298.918,E2 27298.918} C_VEL
LIN {X 0,Y 571.735,Z 826.446,A -85,B 0,C 180,E1 27298.06,E2 27298.06} C_VEL
LIN {X 0,Y 571.221,Z 845.789,A -85,B 0,C 180,E1 27297.069,E2 27297.069} C_VEL
LIN {X 0,Y 570.706,Z 866.154,A -85,B 0,C 180,E1 27295.821,E2 27295.821} C_VEL
LIN {X 0,Y 570.197,Z 885.144,A -85,B 0,C 180,E1 27294.444,E2 27294.444} C_VEL
LIN {X 0,Y 569.697,Z 902.921,A -85,B 0,C 180,E1 27292.929,E2 27292.929} C_VEL
LIN {X 0,Y 569.257,Z 919.534,A -85,B 0,C 180,E1 27291.282,E2 27291.282} C_VEL
LIN {X 0,Y 568.882,Z 935.032,A -85,B 0,C 180,E1 27289.506,E2 27289.506} C_VEL
LIN {X 0,Y 568.569,Z 949.297,A -85,B 0,C 180,E1 27287.611,E2 27287.611} C_VEL
LIN {X 0,Y 568.324,Z 961.475,A -85,B 0,C 180,E1 27285.719,E2 27285.719} C_VEL
LIN {X 0,Y 568.147,Z 972.376,A -85,B 0,C 180,E1 27283.727,E2 27283.727} C_VEL
LIN {X 0,Y 568.035,Z 981.848,A -85,B 0,C 180,E1 27281.678,E2 27281.678} C_VEL
LIN {X 0,Y 567.955,Z 989.533,A -85,B 0,C 180,E1 27279.627,E2 27279.627} C_VEL
LIN {X 0,Y 567.916,Z 995.891,A -85,B 0,C 180,E1 27277.486,E2 27277.486} C_VEL
LIN {X 0,Y 567.911,Z 1000.428,A -85,B 0,C 180,E1 27275.455,E2 27275.455} C_VEL
LIN {X 0,Y 567.914,Z 1003.56,A -85,B 0,C 180,E1 27273.331,E2 27273.331} C_VEL
LIN {X 0,Y 567.914,Z 1005.261,A -85,B 0,C 180,E1 27271.11,E2 27271.11} C_VEL
LIN {X 0,Y 567.907,Z 1005.284,A -85,B 0,C 180,E1 27268.992,E2 27268.992} C_VEL
LIN {X 0,Y 567.908,Z 1003.672,A -85,B 0,C 180,E1 27266.771,E2 27266.771} C_VEL
LIN {X 0,Y 567.905,Z 1000.634,A -85,B 0,C 180,E1 27264.647,E2 27264.647} C_VEL
LIN {X 0,Y 567.912,Z 996.147,A -85,B 0,C 180,E1 27262.617,E2 27262.617} C_VEL
LIN {X 0,Y 567.955,Z 989.888,A -85,B 0,C 180,E1 27260.476,E2 27260.476} C_VEL
LIN {X 0,Y 568.027,Z 982.665,A -85,B 0,C 180,E1 27258.529,E2 27258.529} C_VEL
LIN {X 0,Y 568.139,Z 973.339,A -85,B 0,C 180,E1 27256.465,E2 27256.465} C_VEL
LIN {X 0,Y 568.318,Z 962.75,A -85,B 0,C 180,E1 27254.491,E2 27254.491} C_VEL
LIN {X 0,Y 568.553,Z 950.055,A -85,B 0,C 180,E1 27252.501,E2 27252.501} C_VEL
LIN {X 0,Y 568.858,Z 935.888,A -85,B 0,C 180,E1 27250.6,E2 27250.6} C_VEL
LIN {X 0,Y 569.234,Z 920.217,A -85,B 0,C 180,E1 27248.789,E2 27248.789} C_VEL
LIN {X 0,Y 569.683,Z 903.647,A -85,B 0,C 180,E1 27247.136,E2 27247.136} C_VEL
LIN {X 0,Y 570.178,Z 885.822,A -85,B 0,C 180,E1 27245.611,E2 27245.611} C_VEL
LIN {X 0,Y 570.681,Z 866.907,A -85,B 0,C 180,E1 27244.23,E2 27244.23} C_VEL
LIN {X 0,Y 571.196,Z 846.972,A -85,B 0,C 180,E1 27242.997,E2 27242.997} C_VEL
LIN {X 0,Y 571.693,Z 827.716,A -85,B 0,C 180,E1 27242.001,E2 27242.001} C_VEL
LIN {X 0,Y 572.103,Z 807.109,A -85,B 0,C 180,E1 27241.137,E2 27241.137} C_VEL
LIN {X 0,Y 572.533,Z 784.83,A -85,B 0,C 180,E1 27240.41,E2 27240.41} C_VEL
LIN {X 0,Y 572.826,Z 763.898,A -85,B 0,C 180,E1 27239.912,E2 27239.912} C_VEL
LIN {X 0,Y 573.086,Z 726.265,A -85,B 0,C 180,E1 27239.347,E2 27239.347} C_VEL
LIN {X 0,Y 574.2,Z 492.869,A -85,B 0,C 180,E1 27236.03,E2 27236.03} C_VEL
LIN {X 0,Y 574.206,Z 460.192,A -85,B 0,C 180,E1 27235.546,E2 27235.546} C_VEL
LIN {X 0,Y 573.332,Z 453.785,A -85,B 0,C 180,E1 27235.357,E2 27235.357} C_VEL
LIN {X 0,Y 574.375,Z 395.402,A -85,B 0,C 180,E1 27232.009,E2 27232.009} C_VEL
LIN {X 0,Y 574.613,Z 374.147,A -85,B 0,C 180,E1 27230.743,E2 27230.743} C_VEL
LIN {X 0,Y 569.429,Z 363.375,A -85,B 0,C 180,E1 27229.646,E2 27229.646} C_VEL
LIN {X 0,Y 568.222,Z 360.369,A -85,B 0,C 180,E1 27229.323,E2 27229.323} C_VEL
LIN {X 0,Y 568.181,Z 359.961,A -85,B 0,C 180,E1 27228.981,E2 27228.981} C_VEL
LIN {X 0,Y 568.165,Z 359.962,A -85,B 0,C 180,E1 27225.688,E2 27225.688} C_VEL
LIN {X 0,Y 568.191,Z 359.955,A -85,B 0,C 180,E1 27222.648,E2 27222.648} C_VEL
LIN {X 0,Y 568.155,Z 359.957,A -85,B 0,C 180,E1 27219.423,E2 27219.423} C_VEL
LIN {X 0,Y 568.196,Z 359.955,A -85,B 0,C 180,E1 27216.371,E2 27216.371} C_VEL
LIN {X 0,Y 568.147,Z 359.96,A -85,B 0,C 180,E1 27213.183,E2 27213.183} C_VEL
LIN {X 0,Y 568.213,Z 359.947,A -85,B 0,C 180,E1 27210.042,E2 27210.042} C_VEL
LIN {X 0,Y 568.139,Z 359.96,A -85,B 0,C 180,E1 27206.854,E2 27206.854} C_VEL
LIN {X 0,Y 568.215,Z 359.946,A -85,B 0,C 180,E1 27203.763,E2 27203.763} C_VEL
LIN {X 0,Y 568.134,Z 359.96,A -85,B 0,C 180,E1 27200.608,E2 27200.608} C_VEL
LIN {X 0,Y 568.194,Z 359.961,A -85,B 0,C 180,E1 27197.406,E2 27197.406} C_VEL
LIN {X 0,Y 568.131,Z 359.959,A -85,B 0,C 180,E1 27194.368,E2 27194.368} C_VEL
LIN {X 0,Y 568.187,Z 359.958,A -85,B 0,C 180,E1 27191.161,E2 27191.161} C_VEL
LIN {X 0,Y 568.138,Z 359.959,A -85,B 0,C 180,E1 27188.093,E2 27188.093} C_VEL
LIN {X 0,Y 568.176,Z 359.958,A -85,B 0,C 180,E1 27184.845,E2 27184.845} C_VEL
LIN {X 0,Y 568.15,Z 359.957,A -85,B 0,C 180,E1 27181.815,E2 27181.815} C_VEL
LIN {X 0,Y 568.156,Z 359.954,A -85,B 0,C 180,E1 27178.386,E2 27178.386} C_VEL
LIN {X 0,Y 568.178,Z 359.959,A -85,B 0,C 180,E1 27175.357,E2 27175.357} C_VEL
LIN {X 0,Y 568.156,Z 359.957,A -85,B 0,C 180,E1 27172.11,E2 27172.11} C_VEL
LIN {X 0,Y 568.197,Z 359.956,A -85,B 0,C 180,E1 27169.044,E2 27169.044} C_VEL
LIN {X 0,Y 568.157,Z 359.955,A -85,B 0,C 180,E1 27165.827,E2 27165.827} C_VEL
LIN {X 0,Y 568.218,Z 359.959,A -85,B 0,C 180,E1 27162.7,E2 27162.7} C_VEL
LIN {X 0,Y 568.165,Z 359.956,A -85,B 0,C 180,E1 27159.74,E2 27159.74} C_VEL
LIN {X 0,Y 567.175,Z 360.085,A -85,B 0,C 180,E1 27158.964,E2 27158.964} C_VEL
LIN {X 0,Y 560.731,Z 360.891,A -85,B 0,C 180,E1 27156.726,E2 27156.726} C_VEL
LIN {X 0,Y 560.279,Z 360.943,A -85,B 0,C 180,E1 27156.215,E2 27156.215} C_VEL
LIN {X 0,Y 560.232,Z 360.945,A -85,B 0,C 180,E1 27153.043,E2 27153.043} C_VEL
LIN {X 0,Y 560.247,Z 360.94,A -85,B 0,C 180,E1 27149.664,E2 27149.664} C_VEL
LIN {X 0,Y 560.269,Z 360.947,A -85,B 0,C 180,E1 27146.441,E2 27146.441} C_VEL
LIN {X 0,Y 560.235,Z 360.943,A -85,B 0,C 180,E1 27143.154,E2 27143.154} C_VEL
LIN {X 0,Y 560.281,Z 360.943,A -85,B 0,C 180,E1 27139.892,E2 27139.892} C_VEL
LIN {X 0,Y 560.243,Z 360.944,A -85,B 0,C 180,E1 27136.598,E2 27136.598} C_VEL
LIN {X 0,Y 560.263,Z 360.943,A -85,B 0,C 180,E1 27133.253,E2 27133.253} C_VEL
LIN {X 0,Y 560.274,Z 360.941,A -85,B 0,C 180,E1 27129.97,E2 27129.97} C_VEL
LIN {X 0,Y 560.246,Z 360.939,A -85,B 0,C 180,E1 27126.713,E2 27126.713} C_VEL
LIN {X 0,Y 560.277,Z 360.936,A -85,B 0,C 180,E1 27123.461,E2 27123.461} C_VEL
LIN {X 0,Y 560.288,Z 361.194,A -85,B 0,C 180,E1 27122.153,E2 27122.153} C_VEL
LIN {X 0,Y 564.033,Z 372.79,A -85,B 0,C 180,E1 27120.873,E2 27120.873} C_VEL
LIN {X 0,Y 563.933,Z 383.496,A -85,B 0,C 180,E1 27119.996,E2 27119.996} C_VEL
LIN {X 0,Y 565.703,Z 392.948,A -85,B 0,C 180,E1 27119.747,E2 27119.747} C_VEL
LIN {X 0,Y 564.416,Z 643.401,A -85,B 0,C 180,E1 27116.256,E2 27116.256} C_VEL
LIN {X 0,Y 564.111,Z 663.767,A -85,B 0,C 180,E1 27115.788,E2 27115.788} C_VEL
LIN {X 0,Y 563.72,Z 683.921,A -85,B 0,C 180,E1 27115.135,E2 27115.135} C_VEL
LIN {X 0,Y 563.301,Z 703.263,A -85,B 0,C 180,E1 27114.315,E2 27114.315} C_VEL
LIN {X 0,Y 562.827,Z 721.86,A -85,B 0,C 180,E1 27113.335,E2 27113.335} C_VEL
LIN {X 0,Y 562.316,Z 740.447,A -85,B 0,C 180,E1 27112.143,E2 27112.143} C_VEL
LIN {X 0,Y 561.805,Z 757.907,A -85,B 0,C 180,E1 27110.794,E2 27110.794} C_VEL
LIN {X 0,Y 561.359,Z 773.776,A -85,B 0,C 180,E1 27109.345,E2 27109.345} C_VEL
LIN {X 0,Y 560.954,Z 788.726,A -85,B 0,C 180,E1 27107.744,E2 27107.744} C_VEL
LIN {X 0,Y 560.605,Z 803.007,A -85,B 0,C 180,E1 27105.94,E2 27105.94} C_VEL
LIN {X 0,Y 560.339,Z 815.62,A -85,B 0,C 180,E1 27104.043,E2 27104.043} C_VEL
LIN {X 0,Y 560.145,Z 826.618,A -85,B 0,C 180,E1 27102.053,E2 27102.053} C_VEL
LIN {X 0,Y 560.022,Z 835.582,A -85,B 0,C 180,E1 27100.075,E2 27100.075} C_VEL
LIN {X 0,Y 559.961,Z 843.062,A -85,B 0,C 180,E1 27098.005,E2 27098.005} C_VEL
LIN {X 0,Y 559.932,Z 848.65,A -85,B 0,C 180,E1 27095.942,E2 27095.942} C_VEL
LIN {X 0,Y 559.918,Z 852.516,A -85,B 0,C 180,E1 27093.89,E2 27093.89} C_VEL
LIN {X 0,Y 559.909,Z 854.845,A -85,B 0,C 180,E1 27091.739,E2 27091.739} C_VEL
LIN {X 0,Y 559.904,Z 855.449,A -85,B 0,C 180,E1 27089.693,E2 27089.693} C_VEL
LIN {X 0,Y 559.906,Z 854.494,A -85,B 0,C 180,E1 27087.646,E2 27087.646} C_VEL
LIN {X 0,Y 559.914,Z 851.702,A -85,B 0,C 180,E1 27085.494,E2 27085.494} C_VEL
LIN {X 0,Y 559.935,Z 847.35,A -85,B 0,C 180,E1 27083.438,E2 27083.438} C_VEL
LIN {X 0,Y 559.976,Z 841.275,A -85,B 0,C 180,E1 27081.374,E2 27081.374} C_VEL
LIN {X 0,Y 560.053,Z 833.8,A -85,B 0,C 180,E1 27079.405,E2 27079.405} C_VEL
LIN {X 0,Y 560.194,Z 824.459,A -85,B 0,C 180,E1 27077.424,E2 27077.424} C_VEL
LIN {X 0,Y 560.378,Z 813.598,A -85,B 0,C 180,E1 27075.536,E2 27075.536} C_VEL
LIN {X 0,Y 560.647,Z 801.328,A -85,B 0,C 180,E1 27073.741,E2 27073.741} C_VEL
LIN {X 0,Y 560.983,Z 787.641,A -85,B 0,C 180,E1 27072.042,E2 27072.042} C_VEL
LIN {X 0,Y 561.406,Z 772.235,A -85,B 0,C 180,E1 27070.415,E2 27070.415} C_VEL
LIN {X 0,Y 561.868,Z 755.69,A -85,B 0,C 180,E1 27068.935,E2 27068.935} C_VEL
LIN {X 0,Y 562.371,Z 737.951,A -85,B 0,C 180,E1 27067.597,E2 27067.597} C_VEL
LIN {X 0,Y 562.881,Z 719.404,A -85,B 0,C 180,E1 27066.432,E2 27066.432} C_VEL
LIN {X 0,Y 563.375,Z 700.542,A -85,B 0,C 180,E1 27065.464,E2 27065.464} C_VEL
LIN {X 0,Y 563.79,Z 681.101,A -85,B 0,C 180,E1 27064.671,E2 27064.671} C_VEL
LIN {X 0,Y 564.142,Z 660.727,A -85,B 0,C 180,E1 27064.041,E2 27064.041} C_VEL
LIN {X 0,Y 564.439,Z 639.496,A -85,B 0,C 180,E1 27063.591,E2 27063.591} C_VEL
LIN {X 0,Y 565.695,Z 391.792,A -85,B 0,C 180,E1 27060.146,E2 27060.146} C_VEL
LIN {X 0,Y 563.857,Z 382.824,A -85,B 0,C 180,E1 27059.882,E2 27059.882} C_VEL
LIN {X 0,Y 563.986,Z 372.454,A -85,B 0,C 180,E1 27059.005,E2 27059.005} C_VEL
LIN {X 0,Y 560.297,Z 361.226,A -85,B 0,C 180,E1 27057.756,E2 27057.756} C_VEL
LIN {X 0,Y 560.253,Z 360.943,A -85,B 0,C 180,E1 27055.302,E2 27055.302} C_VEL
LIN {X 0,Y 560.272,Z 360.94,A -85,B 0,C 180,E1 27051.907,E2 27051.907} C_VEL
LIN {X 0,Y 560.283,Z 360.93,A -85,B 0,C 180,E1 27048.547,E2 27048.547} C_VEL
LIN {X 0,Y 560.245,Z 360.939,A -85,B 0,C 180,E1 27045.26,E2 27045.26} C_VEL
LIN {X 0,Y 560.279,Z 360.944,A -85,B 0,C 180,E1 27042.007,E2 27042.007} C_VEL
LIN {X 0,Y 560.245,Z 360.929,A -85,B 0,C 180,E1 27038.755,E2 27038.755} C_VEL
LIN {X 0,Y 560.253,Z 360.947,A -85,B 0,C 180,E1 27035.326,E2 27035.326} C_VEL
LIN {X 0,Y 560.281,Z 360.942,A -85,B 0,C 180,E1 27032.007,E2 27032.007} C_VEL
LIN {X 0,Y 560.234,Z 360.946,A -85,B 0,C 180,E1 27028.808,E2 27028.808} C_VEL
LIN {X 0,Y 560.283,Z 360.943,A -85,B 0,C 180,E1 27025.586,E2 27025.586} C_VEL
LIN {X 0,Y 560.23,Z 360.943,A -85,B 0,C 180,E1 27022.343,E2 27022.343} C_VEL
LIN {X 0,Y 560.259,Z 360.945,A -85,B 0,C 180,E1 27019.062,E2 27019.062} C_VEL
LIN {X 0,Y 560.243,Z 360.943,A -85,B 0,C 180,E1 27015.876,E2 27015.876} C_VEL
LIN {X 0,Y 560.226,Z 360.947,A -85,B 0,C 180,E1 27012.536,E2 27012.536} C_VEL
LIN {X 0,Y 560.273,Z 360.941,A -85,B 0,C 180,E1 27009.346,E2 27009.346} C_VEL
LIN {X 0,Y 560.214,Z 360.942,A -85,B 0,C 180,E1 27006.148,E2 27006.148} C_VEL
LIN {X 0,Y 560.279,Z 360.948,A -85,B 0,C 180,E1 27002.967,E2 27002.967} C_VEL
LIN {X 0,Y 560.209,Z 360.947,A -85,B 0,C 180,E1 26999.796,E2 26999.796} C_VEL
LIN {X 0,Y 560.251,Z 360.949,A -85,B 0,C 180,E1 26996.521,E2 26996.521} C_VEL
LIN {X 0,Y 560.208,Z 360.946,A -85,B 0,C 180,E1 26993.441,E2 26993.441} C_VEL
LIN {X 0,Y 560.214,Z 360.947,A -85,B 0,C 180,E1 26990.031,E2 26990.031} C_VEL
LIN {X 0,Y 560.213,Z 360.948,A -85,B 0,C 180,E1 26987.109,E2 26987.109} C_VEL
LIN {X 0,Y 560.199,Z 360.949,A -85,B 0,C 180,E1 26983.727,E2 26983.727} C_VEL
LIN {X 0,Y 560.231,Z 360.947,A -85,B 0,C 180,E1 26980.721,E2 26980.721} C_VEL
LIN {X 0,Y 560.198,Z 360.944,A -85,B 0,C 180,E1 26977.435,E2 26977.435} C_VEL
LIN {X 0,Y 560.265,Z 360.94,A -85,B 0,C 180,E1 26974.3,E2 26974.3} C_VEL
LIN {X 0,Y 560.201,Z 360.946,A -85,B 0,C 180,E1 26971.074,E2 26971.074} C_VEL
LIN {X 0,Y 560.278,Z 360.944,A -85,B 0,C 180,E1 26967.951,E2 26967.951} C_VEL
LIN {X 0,Y 560.209,Z 360.942,A -85,B 0,C 180,E1 26964.796,E2 26964.796} C_VEL
LIN {X 0,Y 560.261,Z 360.944,A -85,B 0,C 180,E1 26961.571,E2 26961.571} C_VEL
LIN {X 0,Y 560.216,Z 360.947,A -85,B 0,C 180,E1 26958.536,E2 26958.536} C_VEL
LIN {X 0,Y 560.242,Z 360.945,A -85,B 0,C 180,E1 26955.175,E2 26955.175} C_VEL
LIN {X 0,Y 560.239,Z 360.936,A -85,B 0,C 180,E1 26952.061,E2 26952.061} C_VEL
LIN {X 0,Y 560.318,Z 361.257,A -85,B 0,C 180,E1 26951.301,E2 26951.301} C_VEL
LIN {X 0,Y 561.515,Z 364.39,A -85,B 0,C 180,E1 26950.976,E2 26950.976} C_VEL
LIN {X 0,Y 568.19,Z 378.167,A -85,B 0,C 180,E1 26949.539,E2 26949.539} C_VEL
LIN {X 0,Y 566.999,Z 429.468,A -85,B 0,C 180,E1 26946.52,E2 26946.52} C_VEL
LIN {X 0,Y 566.633,Z 455.335,A -85,B 0,C 180,E1 26945.057,E2 26945.057} C_VEL
LIN {X 0,Y 567.771,Z 464.244,A -85,B 0,C 180,E1 26944.839,E2 26944.839} C_VEL
LIN {X 0,Y 566.403,Z 690.393,A -85,B 0,C 180,E1 26941.576,E2 26941.576} C_VEL
LIN {X 0,Y 565.937,Z 762.32,A -85,B 0,C 180,E1 26940.527,E2 26940.527} C_VEL
LIN {X 0,Y 565.546,Z 783.746,A -85,B 0,C 180,E1 26940.023,E2 26940.023} C_VEL
LIN {X 0,Y 565.071,Z 805.899,A -85,B 0,C 180,E1 26939.304,E2 26939.304} C_VEL
LIN {X 0,Y 564.575,Z 826.445,A -85,B 0,C 180,E1 26938.448,E2 26938.448} C_VEL
LIN {X 0,Y 563.935,Z 846.787,A -85,B 0,C 180,E1 26937.391,E2 26937.391} C_VEL
LIN {X 0,Y 563.301,Z 867.176,A -85,B 0,C 180,E1 26936.114,E2 26936.114} C_VEL
LIN {X 0,Y 562.698,Z 885.386,A -85,B 0,C 180,E1 26934.771,E2 26934.771} C_VEL
LIN {X 0,Y 562.102,Z 903.23,A -85,B 0,C 180,E1 26933.229,E2 26933.229} C_VEL
LIN {X 0,Y 561.573,Z 919.703,A -85,B 0,C 180,E1 26931.57,E2 26931.57} C_VEL
LIN {X 0,Y 561.086,Z 935.883,A -85,B 0,C 180,E1 26929.68,E2 26929.68} C_VEL
LIN {X 0,Y 560.702,Z 950.051,A -85,B 0,C 180,E1 26927.753,E2 26927.753} C_VEL
LIN {X 0,Y 560.407,Z 962.743,A -85,B 0,C 180,E1 26925.734,E2 26925.734} C_VEL
LIN {X 0,Y 560.193,Z 973.337,A -85,B 0,C 180,E1 26923.731,E2 26923.731} C_VEL
LIN {X 0,Y 560.051,Z 983.071,A -85,B 0,C 180,E1 26921.533,E2 26921.533} C_VEL
LIN {X 0,Y 559.967,Z 990.593,A -85,B 0,C 180,E1 26919.454,E2 26919.454} C_VEL
LIN {X 0,Y 559.917,Z 996.4,A -85,B 0,C 180,E1 26917.387,E2 26917.387} C_VEL
LIN {X 0,Y 559.905,Z 1000.824,A -85,B 0,C 180,E1 26915.328,E2 26915.328} C_VEL
LIN {X 0,Y 559.904,Z 1003.785,A -85,B 0,C 180,E1 26913.173,E2 26913.173} C_VEL
LIN {X 0,Y 559.904,Z 1005.306,A -85,B 0,C 180,E1 26910.921,E2 26910.921} C_VEL
LIN {X 0,Y 559.91,Z 1005.238,A -85,B 0,C 180,E1 26908.773,E2 26908.773} C_VEL
LIN {X 0,Y 559.915,Z 1003.514,A -85,B 0,C 180,E1 26906.58,E2 26906.58} C_VEL
LIN {X 0,Y 559.922,Z 1000.222,A -85,B 0,C 180,E1 26904.365,E2 26904.365} C_VEL
LIN {X 0,Y 559.933,Z 995.639,A -85,B 0,C 180,E1 26902.305,E2 26902.305} C_VEL
LIN {X 0,Y 559.979,Z 989.18,A -85,B 0,C 180,E1 26900.132,E2 26900.132} C_VEL
LIN {X 0,Y 560.076,Z 981.398,A -85,B 0,C 180,E1 26898.041,E2 26898.041} C_VEL
LIN {X 0,Y 560.223,Z 971.782,A -85,B 0,C 180,E1 26895.954,E2 26895.954} C_VEL
LIN {X 0,Y 560.456,Z 960.204,A -85,B 0,C 180,E1 26893.843,E2 26893.843} C_VEL
LIN {X 0,Y 560.77,Z 947.456,A -85,B 0,C 180,E1 26891.867,E2 26891.867} C_VEL
LIN {X 0,Y 561.163,Z 933.339,A -85,B 0,C 180,E1 26889.998,E2 26889.998} C_VEL
LIN {X 0,Y 561.62,Z 918.192,A -85,B 0,C 180,E1 26888.268,E2 26888.268} C_VEL
LIN {X 0,Y 562.188,Z 900.517,A -85,B 0,C 180,E1 26886.526,E2 26886.526} C_VEL
LIN {X 0,Y 562.768,Z 883.066,A -85,B 0,C 180,E1 26885.045,E2 26885.045} C_VEL
LIN {X 0,Y 563.416,Z 863.949,A -85,B 0,C 180,E1 26883.666,E2 26883.666} C_VEL
LIN {X 0,Y 563.999,Z 844.815,A -85,B 0,C 180,E1 26882.499,E2 26882.499} C_VEL
LIN {X 0,Y 564.595,Z 825.212,A -85,B 0,C 180,E1 26881.497,E2 26881.497} C_VEL
LIN {X 0,Y 565.107,Z 804.844,A -85,B 0,C 180,E1 26880.656,E2 26880.656} C_VEL
LIN {X 0,Y 565.558,Z 782.617,A -85,B 0,C 180,E1 26879.946,E2 26879.946} C_VEL
LIN {X 0,Y 565.947,Z 760.99,A -85,B 0,C 180,E1 26879.451,E2 26879.451} C_VEL
LIN {X 0,Y 567.307,Z 536.635,A -85,B 0,C 180,E1 26876.215,E2 26876.215} C_VEL
LIN {X 0,Y 567.595,Z 461.545,A -85,B 0,C 180,E1 26875.107,E2 26875.107} C_VEL
LIN {X 0,Y 566.53,Z 453.812,A -85,B 0,C 180,E1 26874.88,E2 26874.88} C_VEL
LIN {X 0,Y 567.759,Z 396.75,A -85,B 0,C 180,E1 26871.568,E2 26871.568} C_VEL
LIN {X 0,Y 568.015,Z 377.745,A -85,B 0,C 180,E1 26870.421,E2 26870.421} C_VEL
LIN {X 0,Y 561.515,Z 364.389,A -85,B 0,C 180,E1 26869.024,E2 26869.024} C_VEL
LIN {X 0,Y 560.308,Z 361.19,A -85,B 0,C 180,E1 26868.686,E2 26868.686} C_VEL
LIN {X 0,Y 560.218,Z 360.951,A -85,B 0,C 180,E1 26865.466,E2 26865.466} C_VEL
LIN {X 0,Y 560.279,Z 360.947,A -85,B 0,C 180,E1 26862.225,E2 26862.225} C_VEL
LIN {X 0,Y 560.213,Z 360.945,A -85,B 0,C 180,E1 26859.052,E2 26859.052} C_VEL
LIN {X 0,Y 560.255,Z 360.937,A -85,B 0,C 180,E1 26855.828,E2 26855.828} C_VEL
LIN {X 0,Y 560.213,Z 360.949,A -85,B 0,C 180,E1 26852.737,E2 26852.737} C_VEL
LIN {X 0,Y 560.224,Z 360.946,A -85,B 0,C 180,E1 26849.393,E2 26849.393} C_VEL
LIN {X 0,Y 560.219,Z 360.948,A -85,B 0,C 180,E1 26846.382,E2 26846.382} C_VEL
LIN {X 0,Y 560.204,Z 360.944,A -85,B 0,C 180,E1 26843.009,E2 26843.009} C_VEL
LIN {X 0,Y 560.228,Z 360.949,A -85,B 0,C 180,E1 26840.039,E2 26840.039} C_VEL
LIN {X 0,Y 560.199,Z 360.949,A -85,B 0,C 180,E1 26836.806,E2 26836.806} C_VEL
LIN {X 0,Y 560.227,Z 360.948,A -85,B 0,C 180,E1 26833.836,E2 26833.836} C_VEL
LIN {X 0,Y 560.199,Z 360.947,A -85,B 0,C 180,E1 26830.593,E2 26830.593} C_VEL
LIN {X 0,Y 560.254,Z 360.948,A -85,B 0,C 180,E1 26827.485,E2 26827.485} C_VEL
LIN {X 0,Y 560.202,Z 360.948,A -85,B 0,C 180,E1 26824.299,E2 26824.299} C_VEL
LIN {X 0,Y 560.28,Z 360.948,A -85,B 0,C 180,E1 26821.125,E2 26821.125} C_VEL
LIN {X 0,Y 560.206,Z 360.943,A -85,B 0,C 180,E1 26817.954,E2 26817.954} C_VEL
LIN {X 0,Y 560.262,Z 360.941,A -85,B 0,C 180,E1 26814.694,E2 26814.694} C_VEL
LIN {X 0,Y 560.217,Z 360.947,A -85,B 0,C 180,E1 26811.584,E2 26811.584} C_VEL
LIN {X 0,Y 560.239,Z 360.945,A -85,B 0,C 180,E1 26808.261,E2 26808.261} C_VEL
LIN {X 0,Y 560.235,Z 360.945,A -85,B 0,C 180,E1 26805.214,E2 26805.214} C_VEL
LIN {X 0,Y 560.225,Z 360.944,A -85,B 0,C 180,E1 26801.8,E2 26801.8} C_VEL
LIN {X 0,Y 560.278,Z 360.949,A -85,B 0,C 180,E1 26798.65,E2 26798.65} C_VEL
LIN {X 0,Y 560.279,Z 360.943,A -85,B 0,C 180,E1 26796.215,E2 26796.215} C_VEL
LIN {X 0,Y 559.249,Z 361.068,A -85,B 0,C 180,E1 26795.428,E2 26795.428} C_VEL
LIN {X 0,Y 552.812,Z 361.872,A -85,B 0,C 180,E1 26793.216,E2 26793.216} C_VEL
LIN {X 0,Y 552.325,Z 361.933,A -85,B 0,C 180,E1 26792.641,E2 26792.641} C_VEL
LIN {X 0,Y 552.292,Z 361.93,A -85,B 0,C 180,E1 26789.298,E2 26789.298} C_VEL
LIN {X 0,Y 552.342,Z 361.931,A -85,B 0,C 180,E1 26786.113,E2 26786.113} C_VEL
LIN {X 0,Y 552.296,Z 361.934,A -85,B 0,C 180,E1 26782.925,E2 26782.925} C_VEL
LIN {X 0,Y 552.34,Z 361.93,A -85,B 0,C 180,E1 26779.604,E2 26779.604} C_VEL
LIN {X 0,Y 552.326,Z 361.925,A -85,B 0,C 180,E1 26776.238,E2 26776.238} C_VEL
LIN {X 0,Y 552.304,Z 361.934,A -85,B 0,C 180,E1 26772.892,E2 26772.892} C_VEL
LIN {X 0,Y 552.341,Z 361.934,A -85,B 0,C 180,E1 26769.705,E2 26769.705} C_VEL
LIN {X 0,Y 552.307,Z 361.929,A -85,B 0,C 180,E1 26766.422,E2 26766.422} C_VEL
LIN {X 0,Y 552.335,Z 361.928,A -85,B 0,C 180,E1 26763.012,E2 26763.012} C_VEL
LIN {X 0,Y 552.373,Z 362.347,A -85,B 0,C 180,E1 26762.578,E2 26762.578} C_VEL
LIN {X 0,Y 556.734,Z 375.825,A -85,B 0,C 180,E1 26761.056,E2 26761.056} C_VEL
LIN {X 0,Y 556.669,Z 383.466,A -85,B 0,C 180,E1 26760.43,E2 26760.43} C_VEL
LIN {X 0,Y 558.751,Z 394.336,A -85,B 0,C 180,E1 26760.136,E2 26760.136} C_VEL
LIN {X 0,Y 557.241,Z 643.23,A -85,B 0,C 180,E1 26756.624,E2 26756.624} C_VEL
LIN {X 0,Y 556.886,Z 663.556,A -85,B 0,C 180,E1 26756.154,E2 26756.154} C_VEL
LIN {X 0,Y 556.452,Z 683.201,A -85,B 0,C 180,E1 26755.515,E2 26755.515} C_VEL
LIN {X 0,Y 555.937,Z 703.275,A -85,B 0,C 180,E1 26754.658,E2 26754.658} C_VEL
LIN {X 0,Y 555.371,Z 721.869,A -85,B 0,C 180,E1 26753.668,E2 26753.668} C_VEL
LIN {X 0,Y 554.772,Z 740.456,A -85,B 0,C 180,E1 26752.46,E2 26752.46} C_VEL
LIN {X 0,Y 554.181,Z 757.852,A -85,B 0,C 180,E1 26751.099,E2 26751.099} C_VEL
LIN {X 0,Y 553.649,Z 773.784,A -85,B 0,C 180,E1 26749.625,E2 26749.625} C_VEL
LIN {X 0,Y 553.162,Z 788.731,A -85,B 0,C 180,E1 26748.002,E2 26748.002} C_VEL
LIN {X 0,Y 552.749,Z 803.011,A -85,B 0,C 180,E1 26746.173,E2 26746.173} C_VEL
LIN {X 0,Y 552.425,Z 815.626,A -85,B 0,C 180,E1 26744.248,E2 26744.248} C_VEL
LIN {X 0,Y 552.2,Z 826.623,A -85,B 0,C 180,E1 26742.229,E2 26742.229} C_VEL
LIN {X 0,Y 552.049,Z 835.586,A -85,B 0,C 180,E1 26740.222,E2 26740.222} C_VEL
LIN {X 0,Y 551.973,Z 843.065,A -85,B 0,C 180,E1 26738.121,E2 26738.121} C_VEL
LIN {X 0,Y 551.933,Z 848.756,A -85,B 0,C 180,E1 26735.986,E2 26735.986} C_VEL
LIN {X 0,Y 551.919,Z 852.517,A -85,B 0,C 180,E1 26733.947,E2 26733.947} C_VEL
LIN {X 0,Y 551.909,Z 854.846,A -85,B 0,C 180,E1 26731.764,E2 26731.764} C_VEL
LIN {X 0,Y 551.904,Z 855.449,A -85,B 0,C 180,E1 26729.688,E2 26729.688} C_VEL
LIN {X 0,Y 551.906,Z 854.493,A -85,B 0,C 180,E1 26727.612,E2 26727.612} C_VEL
LIN {X 0,Y 551.915,Z 851.7,A -85,B 0,C 180,E1 26725.428,E2 26725.428} C_VEL
LIN {X 0,Y 551.94,Z 847.348,A -85,B 0,C 180,E1 26723.343,E2 26723.343} C_VEL
LIN {X 0,Y 551.987,Z 841.273,A -85,B 0,C 180,E1 26721.249,E2 26721.249} C_VEL
LIN {X 0,Y 552.077,Z 833.796,A -85,B 0,C 180,E1 26719.25,E2 26719.25} C_VEL
LIN {X 0,Y 552.248,Z 824.456,A -85,B 0,C 180,E1 26717.24,E2 26717.24} C_VEL
LIN {X 0,Y 552.474,Z 813.595,A -85,B 0,C 180,E1 26715.324,E2 26715.324} C_VEL
LIN {X 0,Y 552.794,Z 801.324,A -85,B 0,C 180,E1 26713.504,E2 26713.504} C_VEL
LIN {X 0,Y 553.195,Z 787.634,A -85,B 0,C 180,E1 26711.78,E2 26711.78} C_VEL
LIN {X 0,Y 553.707,Z 771.923,A -85,B 0,C 180,E1 26710.101,E2 26710.101} C_VEL
LIN {X 0,Y 554.282,Z 754.832,A -85,B 0,C 180,E1 26708.561,E2 26708.561} C_VEL
LIN {X 0,Y 554.884,Z 736.942,A -85,B 0,C 180,E1 26707.208,E2 26707.208} C_VEL
LIN {X 0,Y 555.464,Z 718.526,A -85,B 0,C 180,E1 26706.048,E2 26706.048} C_VEL
LIN {X 0,Y 556.051,Z 699.374,A -85,B 0,C 180,E1 26705.063,E2 26705.063} C_VEL
LIN {X 0,Y 556.558,Z 679.598,A -85,B 0,C 180,E1 26704.261,E2 26704.261} C_VEL
LIN {X 0,Y 556.95,Z 659.633,A -85,B 0,C 180,E1 26703.651,E2 26703.651} C_VEL
LIN {X 0,Y 557.272,Z 638.598,A -85,B 0,C 180,E1 26703.21,E2 26703.21} C_VEL
LIN {X 0,Y 558.76,Z 393.349,A -85,B 0,C 180,E1 26699.76,E2 26699.76} C_VEL
LIN {X 0,Y 556.599,Z 382.828,A -85,B 0,C 180,E1 26699.447,E2 26699.447} C_VEL
LIN {X 0,Y 556.599,Z 374.947,A -85,B 0,C 180,E1 26698.768,E2 26698.768} C_VEL
LIN {X 0,Y 552.37,Z 362.287,A -85,B 0,C 180,E1 26697.321,E2 26697.321} C_VEL
LIN {X 0,Y 552.335,Z 361.923,A -85,B 0,C 180,E1 26696.491,E2 26696.491} C_VEL
LIN {X 0,Y 552.316,Z 361.924,A -85,B 0,C 180,E1 26693.145,E2 26693.145} C_VEL
LIN {X 0,Y 552.324,Z 361.926,A -85,B 0,C 180,E1 26689.744,E2 26689.744} C_VEL
LIN {X 0,Y 552.342,Z 361.932,A -85,B 0,C 180,E1 26686.393,E2 26686.393} C_VEL
LIN {X 0,Y 552.305,Z 361.932,A -85,B 0,C 180,E1 26683.156,E2 26683.156} C_VEL
